// TwinCAT 3 PLC project x_template_xPlc
// Title: x_template_xPlc
// Company: TcOpen.MTS
// ProjectVersion: 0.6.0.913
// ProgramVersion: 3.1.4023.0
// libraries:
//   Tc2_Standard, * (Beckhoff Automation GmbH)
//   Tc2_System, * (Beckhoff Automation GmbH)
//   Tc3_Module, * (Beckhoff Automation GmbH)
//   TcoAbbRobotics, 0.11.0.68 (Vortex.Library)
//   TcoAbstractions, 0.11.0.68 (Vortex.Library)
//   TcoAimTtiPowerSupply, 0.11.0.68 (Vortex.Library)
//   TcoCognexVision, 0.11.0.68 (Vortex.Library)
//   TcoCore, 0.11.0.68 (Vortex.Library)
//   TcoData, 0.11.0.68 (Vortex.Library)
//   TcoDrivesBeckhoff, 0.11.0.68 (Vortex.Library)
//   TcoElements, 0.11.0.68 (Vortex.Library)
//   TcoInspectors, 0.11.0.68 (Vortex.Library)
//   TcoIo, 0.11.0.68 (Vortex.Library)
//   TcoKukaRobotics, 0.11.0.68 (Vortex.Library)
//   TcoMitsubishiRobotics, 0.11.0.68 (Vortex.Library)
//   TcoPneumatics, 0.11.0.68 (Vortex.Library)
//   TcoRexrothPress, 0.11.0.68 (Vortex.Library)
//   TcoTixonFeeding, 0.11.0.68 (Vortex.Library)
//   TcoUrRobotics, 0.11.0.68 (Vortex.Library)
//   TcoUtilities, 0.11.0.68 (Vortex.Library)
// project tree:
//   Abstractions/Components/ArrayRenderingExample/ SampleArrayToRender.TcDUT (not stored), SampleDataItem.TcDUT (not stored)
//   Abstractions/Components/MtsFeeding/ TcoFeedingSequenceTask.TcPOU, TcoPlsPaletizator.TcPOU, TcoPlsPaletizator_Components.TcDUT, TcoPlsPaletizator_Config_v_1_x_x.TcDUT, TcoPlsPaletizator_Control_v_1_x_x.TcDUT (not stored), TcoPlsPaletizator_Status_v_1_x_x.TcDUT
//   Abstractions/Components/WrappedComponent/ WrappedComponentExample.TcPOU (not stored), WrappedComponentExample_Config.TcDUT (not stored), WrappedComponentExample_Control.TcDUT (not stored), WrappedComponentExample_Status.TcDUT (not stored), WrappedComponentsExample.TcDUT (not stored)
//   Abstractions/CUBase/ CuBaseRecurringFail.TcDUT (not stored), CuBaseRecurringFailures.TcDUT (not stored), CUBase.TcPOU (not stored), CUBaseStatusInfo.TcDUT (not stored), CUBaseSettings.TcDUT (not stored), CUComponentsBase.TcDUT (not stored), ICUBase.TcIO (not stored), ICUTask.TcIO (not stored), OperatorInfo.TcDUT (not stored)
//   Abstractions/CUBase/Data/ CuHeader.TcDUT (not stored), CUProcessDataBase.TcDUT (not stored), CUTechnologicalDataBase.TcDUT (not stored), eCUMode.TcDUT (not stored), eCUState.TcDUT (not stored), eDataEntityInvokeType.TcDUT (not stored), EntityHeader.TcDUT (not stored)
//   Abstractions/CUBase/RemoteTasks/ ProductionPlaner.TcPOU (not stored)
//   Abstractions/CUBase/Tasks/ CUBaseAutomat.TcPOU (not stored), CUBaseSuspend.TcPOU (not stored), CUBaseGround.TcPOU (not stored), CUBaseRecover.TcPOU (not stored)
//   Abstractions/Generic/NotificationPanel/ NotificationPanel.TcPOU (not stored), NotificationPanelInfo.TcDUT (not stored)
//   Abstractions/Generic/TagsPairing/ eTagPairingAnswer.TcDUT (not stored), eTagPairingMode.TcDUT (not stored), eTagPairingStatus.TcDUT (not stored), PairTagTask.TcPOU (not stored), TagsPairing.TcDUT (not stored)
//   Abstractions/Safety/ControlButtons/ TcoControlButtons.TcPOU (not stored), ITcoControlButtons.TcIO (not stored), TcoControledZone_Info.TcDUT (not stored)
//   Abstractions/Safety/ControlledZone/ TcoControlledZoneActionTask.TcPOU (not stored), TcoControlledZone.TcPOU (not stored), TcoControlledZone_Config.TcDUT (not stored), TcoControlledZone_Status.TcDUT (not stored)
//   Abstractions/Safety/ControlVoltage/ ITcoControlVoltage.TcIO (not stored), TcoControlVoltage.TcPOU (not stored)
//   Abstractions/Safety/DoorCircuit/ TcoDoorCircuit_Status.TcDUT (not stored), TcoDoorCircuit_Config.TcDUT (not stored), TcoDoorCircuit.TcPOU (not stored), ITcoDoorCircuit.TcIO (not stored)
//   Abstractions/Safety/Doors/ ITcoDoorLock.TcIO (not stored), TcoStandardDoor.TcPOU (not stored), TcoBasicDoor.TcPOU (not stored)
//   Abstractions/Safety/Estop/ TcoEmergencyStop.TcPOU (not stored)
//   Abstractions/Safety/KeyMode/ TcoKeyMode_Config.TcDUT (not stored), TcoKeyMode_Status.TcDUT (not stored), TcoKeyMode.TcPOU (not stored), ITcoKeyMode.TcIO (not stored)
//   Abstractions/Safety/KeyNormalService/ TcoKeyNormalService.TcPOU (not stored), ITcoKeyNormalSevice.TcIO (not stored)
//   Abstractions/TcoCore/ CycleTimeAnalitics.TcDUT (not stored), TcoInnerTask.TcPOU (not stored), TcoTaskedSequencer.TcPOU (not stored), TcoTaskedService.TcPOU (not stored)
//   Abstractions/Technology/ eStations.TcDUT (not stored)
//   / MAIN.TcPOU (not stored), PlcTask.TcTTO (not stored)
//   Technology/CU00x/Automat/ CU00xAutomatParalell_1_Task.TcPOU (not stored), CU00xAutomatTask.TcPOU (not stored)
//   Technology/CU00x/Components/ CU00xExamplesOfComponents.TcDUT, CU00xComponents.TcDUT
//   Technology/CU00x/Data/ CU00xTechnologicalData.TcDUT (not stored), CU00xDialogContent.TcPOU (not stored), CU00xProcessData.TcDUT (not stored)
//   Technology/CU00x/Ground/ CU00xGroundTask.TcPOU (not stored)
//   Technology/CU00x/Manual/ CU00xManualTask.TcPOU (not stored)
//   Technology/CU00x/Positions/ CU00xTestMultiPositions.TcPOU (not stored), Cu00xTestPositions.TcPOU (not stored)
//   Technology/CU00x/Safety/Suspend/ CU00xSuspendTask.TcPOU
//   Technology/CU00x/Safety/Recover/ CU00xRecoverTask.TcPOU (not stored)
//   Technology/Data/ ProcessData.TcDUT, ProcessDataManager.TcPOU (not stored), TcoEntityBase.TcDUT, TechnologicalDataManager.TcPOU (not stored), TechnologyData.TcDUT
//   Technology/CU00x/ CU00x.TcPOU
//   Technology/ Technology.TcPOU, TechnologyComponents.TcDUT (not stored)
//   DUTs/IO/PDOs/ Device_State_F0482DC3.TcDUT, Device_Control_6258066A.TcDUT, Inputs_23559BB0.TcDUT, Outputs_FC2FACAD.TcDUT, Modules_85784B27.TcDUT, Channel_830843C1.TcDUT, Channel_42CA91F7.TcDUT
//   DUTs/IO/Boxes/ EK1200_013D0B49.TcDUT, EK1122_1FC0878B.TcDUT (not stored), AES_510494FB.TcDUT, EPP1322_1FC0878B.TcDUT, EPP1809_32157CFD.TcDUT, EPP1008_78E8D3DD.TcDUT, EL1809_32157CFD.TcDUT (not stored), EL2809_2B6483BD.TcDUT, EL9011_D65D3D32.TcDUT
//   DUTs/IO/Devices/ SyncUnitTasks_4BE01469.TcDUT, SyncUnits_67D36DDA.TcDUT
//   DUTs/IO/Topology/ EK_E812B8FA.TcDUT, EC_4E5C738F.TcDUT, EC_245FBB9A.TcDUT
//   GVLs/ GVL_iXlinker.TcGVL
// real-time tasks:
//   TASK PlcTask: cycle T#10ms, priority 20, ADS port 350
//   TASK PlcTask1: cycle T#10ms, priority 21, ADS port 351
// I/O:
//   DEVICE EC1 (disabled), AmsNetId 172.20.21.220.7.1
//     (EK1200) [EK1200-5000 EtherCAT Power supply (2A E-Bus)]
//       EC (EK1122) [EK1122 2 port EtherCAT junction]
//       PN (EL6631) [EL6631 PROFINET IO Controller]
//       IA1 (EL1809) [EL1809 16Ch. Dig. Input 24V, 3ms]
//       QA1 (EL2809) [EL2809 16Ch. Dig. Output 24V, 0.5A]
//       Term 6 (EL4004) [EL4004 4Ch. Ana. Output 0-10V, 12bit]
//       Term 7 (EL7342) [EL7342 2Ch. DC motor output stage (50V, 3.5A)]
//       Term 8 (EL4004) [EL4004 4Ch. Ana. Output 0-10V, 12bit]
//       Term 9 (EL6001) [EL6001 Interface (RS232)]
//       Term 13 (EL9011) [EL9011 End Terminal]
//   DEVICE EC (disabled), AmsNetId 172.20.21.220.2.1
//     EC [EK1200-5000 EtherCAT Power supply (2A E-Bus)]
//       EK [EK1122 2 port EtherCAT junction]
//         PNEU [AES Fieldbus Coupler Gen2]
//           modules: Modules
//         AB [EPP1322-0001 3 port EtherCAT P gateway]
//         AB21 [EPP1809-0021 16 Ch. Dig. Input 24V, 3ms, M8]
//         AB22 [EPP1809-0021 16 Ch. Dig. Input 24V, 3ms, M8]
//         AB23 [EPP1008-0001 8 Ch. Dig. Input 24V, 3ms, M8]
//         AB24 [EPP1008-0001 8 Ch. Dig. Input 24V, 3ms, M8]
//       IA1 [EL1809 16Ch. Dig. Input 24V, 3ms]
//       QA1 [EL2809-0015 16Ch. Dig. Output 24V DC, 0.35A, not short-circuit proof]
//       Term 11 (EL9011) [EL9011 End Terminal]
// variable links:
//   x_template_xPlc/x_template_xPlc Instance <-> EC
//     PlcTask Inputs/GVL_iXlinker.EC.InfoData.AmsNetId <-> InfoData/AmsNetId
//     PlcTask Inputs/GVL_iXlinker.EC.InfoData.CfgSlaveCount <-> InfoData/CfgSlaveCount
//     PlcTask Inputs/GVL_iXlinker.EC.InfoData.ChangeCount <-> InfoData/ChangeCount
//     PlcTask Inputs/GVL_iXlinker.EC.InfoData.DevId <-> InfoData/DevId
//     PlcTask Inputs/GVL_iXlinker.EC.Inputs.DevState <-> Inputs/DevState
//     PlcTask Inputs/GVL_iXlinker.EC.Inputs.Frm0InputToggle <-> Inputs/Frm0InputToggle
//     PlcTask Inputs/GVL_iXlinker.EC.Inputs.Frm0State <-> Inputs/Frm0State
//     PlcTask Inputs/GVL_iXlinker.EC.Inputs.Frm0WcState <-> Inputs/Frm0WcState
//     PlcTask Inputs/GVL_iXlinker.EC.Inputs.SlaveCount <-> Inputs/SlaveCount
//     PlcTask Inputs/GVL_iXlinker.EC.SyncUnits._default.PlcTask.InfoData.ObjectId <-> SyncUnits/<default>/PlcTask/InfoData/ObjectId
//     PlcTask Inputs/GVL_iXlinker.EC.SyncUnits._default.PlcTask.InfoData.SlaveCount <-> SyncUnits/<default>/PlcTask/InfoData/SlaveCount
//     PlcTask Inputs/GVL_iXlinker.EC.SyncUnits._default.PlcTask.InfoData.State <-> SyncUnits/<default>/PlcTask/InfoData/State
//     PlcTask Inputs/GVL_iXlinker.EC.SyncUnits._default.PlcTask.WcState.WcState <-> SyncUnits/<default>/PlcTask/WcState/WcState
//     PlcTask Outputs/GVL_iXlinker.EC.Outputs.DevCtrl <-> Outputs/DevCtrl
//     PlcTask Outputs/GVL_iXlinker.EC.Outputs.Frm0Ctrl <-> Outputs/Frm0Ctrl
//     PlcTask Outputs/GVL_iXlinker.EC.Outputs.Frm0WcCtrl <-> Outputs/Frm0WcCtrl
//   x_template_xPlc/x_template_xPlc Instance <-> EC/EC/EK
//     PlcTask Inputs/GVL_iXlinker.EC.EC.EK.InfoData.State <-> InfoData/State
//   x_template_xPlc/x_template_xPlc Instance <-> EC/EC/EK/AB
//     PlcTask Inputs/GVL_iXlinker.EC.EC.EK.AB.InfoData.State <-> InfoData/State
//   x_template_xPlc/x_template_xPlc Instance <-> EC/EC/EK/AB21
//     PlcTask Inputs/GVL_iXlinker.EC.EC.EK.AB21.Channel_{1..16}.Input <-> Channel {1..16}/Input  (16 links)
//     PlcTask Inputs/GVL_iXlinker.EC.EC.EK.AB21.InfoData.State <-> InfoData/State
//     PlcTask Inputs/GVL_iXlinker.EC.EC.EK.AB21.WcState.InputToggle <-> WcState/InputToggle
//     PlcTask Inputs/GVL_iXlinker.EC.EC.EK.AB21.WcState.WcState <-> WcState/WcState
//   x_template_xPlc/x_template_xPlc Instance <-> EC/EC/EK/AB22
//     PlcTask Inputs/GVL_iXlinker.EC.EC.EK.AB22.Channel_{1..16}.Input <-> Channel {1..16}/Input  (16 links)
//     PlcTask Inputs/GVL_iXlinker.EC.EC.EK.AB22.InfoData.State <-> InfoData/State
//     PlcTask Inputs/GVL_iXlinker.EC.EC.EK.AB22.WcState.InputToggle <-> WcState/InputToggle
//     PlcTask Inputs/GVL_iXlinker.EC.EC.EK.AB22.WcState.WcState <-> WcState/WcState
//   x_template_xPlc/x_template_xPlc Instance <-> EC/EC/EK/AB23
//     PlcTask Inputs/GVL_iXlinker.EC.EC.EK.AB23.Channel_{1..8}.Input <-> Channel {1..8}/Input  (8 links)
//     PlcTask Inputs/GVL_iXlinker.EC.EC.EK.AB23.InfoData.State <-> InfoData/State
//     PlcTask Inputs/GVL_iXlinker.EC.EC.EK.AB23.WcState.InputToggle <-> WcState/InputToggle
//     PlcTask Inputs/GVL_iXlinker.EC.EC.EK.AB23.WcState.WcState <-> WcState/WcState
//   x_template_xPlc/x_template_xPlc Instance <-> EC/EC/EK/AB24
//     PlcTask Inputs/GVL_iXlinker.EC.EC.EK.AB24.Channel_{1..8}.Input <-> Channel {1..8}/Input  (8 links)
//     PlcTask Inputs/GVL_iXlinker.EC.EC.EK.AB24.InfoData.State <-> InfoData/State
//     PlcTask Inputs/GVL_iXlinker.EC.EC.EK.AB24.WcState.InputToggle <-> WcState/InputToggle
//     PlcTask Inputs/GVL_iXlinker.EC.EC.EK.AB24.WcState.WcState <-> WcState/WcState
//   x_template_xPlc/x_template_xPlc Instance <-> EC/EC/EK/PNEU
//     PlcTask Inputs/GVL_iXlinker.EC.EC.EK.PNEU.Device_State.CommonValve <-> Device_State/CommonValve
//     PlcTask Inputs/GVL_iXlinker.EC.EC.EK.PNEU.Device_State.Configuration_Error_IO_Module <-> Device_State/Configuration Error IO-Module
//     PlcTask Inputs/GVL_iXlinker.EC.EC.EK.PNEU.Device_State.Configuration_Error_Valve <-> Device_State/Configuration Error Valve
//     PlcTask Inputs/GVL_iXlinker.EC.EC.EK.PNEU.Device_State.Configuratipn_Error_SLS <-> Device_State/Configuratipn Error SLS
//     PlcTask Inputs/GVL_iXlinker.EC.EC.EK.PNEU.Device_State.Count_IO_Module_to_big <-> Device_State/Count IO-Module to big
//     PlcTask Inputs/GVL_iXlinker.EC.EC.EK.PNEU.Device_State.Heardbeat_x <-> Device_State/Heardbeat
//     PlcTask Inputs/GVL_iXlinker.EC.EC.EK.PNEU.Device_State.IO_1_8 <-> Device_State/IO:1-8
//     PlcTask Inputs/GVL_iXlinker.EC.EC.EK.PNEU.Device_State.IO_9_10 <-> Device_State/IO:9-10
//     PlcTask Inputs/GVL_iXlinker.EC.EC.EK.PNEU.Device_State.Switchcounter_Error <-> Device_State/Switchcounter Error
//     PlcTask Inputs/GVL_iXlinker.EC.EC.EK.PNEU.Device_State.UA_OFF <-> Device_State/UA OFF
//     PlcTask Inputs/GVL_iXlinker.EC.EC.EK.PNEU.Device_State.UL_OFF <-> Device_State/UL OFF
//     PlcTask Inputs/GVL_iXlinker.EC.EC.EK.PNEU.Device_State.Undervoltage_5V <-> Device_State/Undervoltage 5V
//     PlcTask Inputs/GVL_iXlinker.EC.EC.EK.PNEU.Device_State.Undervoltage_UA <-> Device_State/Undervoltage UA
//     PlcTask Inputs/GVL_iXlinker.EC.EC.EK.PNEU.Device_State.Undervoltage_UL <-> Device_State/Undervoltage UL
//     PlcTask Inputs/GVL_iXlinker.EC.EC.EK.PNEU.Device_State.Unknown_Module_ID <-> Device_State/Unknown Module ID
//     PlcTask Inputs/GVL_iXlinker.EC.EC.EK.PNEU.Device_State.ValveExtSupplyDiag_1_6 <-> Device_State/ValveExtSupplyDiag:1-6
//     PlcTask Inputs/GVL_iXlinker.EC.EC.EK.PNEU.InfoData.AdsAddr <-> InfoData/AdsAddr
//     PlcTask Inputs/GVL_iXlinker.EC.EC.EK.PNEU.InfoData.State <-> InfoData/State
//     PlcTask Inputs/GVL_iXlinker.EC.EC.EK.PNEU.Modules.Inputs.digital_Data_I[{0..31}] <-> Modules/Inputs/digital Data I_{0..31}  (32 links)
//     PlcTask Inputs/GVL_iXlinker.EC.EC.EK.PNEU.WcState.InputToggle <-> WcState/InputToggle
//     PlcTask Inputs/GVL_iXlinker.EC.EC.EK.PNEU.WcState.WcState <-> WcState/WcState
//     PlcTask Outputs/GVL_iXlinker.EC.EC.EK.PNEU.Device_Control.Default_Modul_Control <-> Device_Control/Default_Modul_Control
//     PlcTask Outputs/GVL_iXlinker.EC.EC.EK.PNEU.Device_Control.Freeze_Output <-> Device_Control/Freeze Output
//     PlcTask Outputs/GVL_iXlinker.EC.EC.EK.PNEU.Device_Control.HL_Swap <-> Device_Control/HL_Swap
//     PlcTask Outputs/GVL_iXlinker.EC.EC.EK.PNEU.Device_Control.Web_App_Disable <-> Device_Control/Web App Disable
//     PlcTask Outputs/GVL_iXlinker.EC.EC.EK.PNEU.Modules.Outputs.digital_Data_O[{0..31}] <-> Modules/Outputs/digital Data O_{0..31}  (32 links)
//   x_template_xPlc/x_template_xPlc Instance <-> EC/EC/IA1
//     PlcTask Inputs/GVL_iXlinker.EC.EC.IA1.Channel_{1..16}.Input <-> Channel {1..16}/Input  (16 links)
//     PlcTask Inputs/GVL_iXlinker.EC.EC.IA1.InfoData.State <-> InfoData/State
//     PlcTask Inputs/GVL_iXlinker.EC.EC.IA1.WcState.InputToggle <-> WcState/InputToggle
//     PlcTask Inputs/GVL_iXlinker.EC.EC.IA1.WcState.WcState <-> WcState/WcState
//   x_template_xPlc/x_template_xPlc Instance <-> EC/EC/QA1
//     PlcTask Inputs/GVL_iXlinker.EC.EC.QA1.InfoData.State <-> InfoData/State
//     PlcTask Inputs/GVL_iXlinker.EC.EC.QA1.WcState.WcState <-> WcState/WcState
//     PlcTask Outputs/GVL_iXlinker.EC.EC.QA1.Channel_{1..16}.Output <-> Channel {1..16}/Output  (16 links)

// ---- Abstractions/Components/MtsFeeding/TcoPlsPaletizator_Components.TcDUT
TYPE TcoPlsPaletizator_Components EXTENDS TcoCore.TcoStruct:
STRUCT
	
	{attribute wpf [Container(Layout.Stack)]}
	{attribute addProperty Name "(I1) <#Pritomnost blistra v presuvaci#>"}
	I1_PresentBlisterEntry : TcoElements.TcoDi(THISSTRUCT);
	
	{attribute addProperty Name "(I2) <#Pritomnost medzery medzi blistrami#>"}
	I2_PresentBlisterEntryEmptySpace : TcoElements.TcoDi(THISSTRUCT);
	
	{attribute addProperty Name "(I3) <#Zasobik blistrov prazdny#>"}
	I3_PresentBlistersInBufferEmpty : TcoElements.TcoDi(THISSTRUCT);

	
	{attribute addProperty Name "(I4) <#Pritomnost blistra v pracovnej pozicii#>"}
	I4_PresentBlisterInWorkingPos : TcoElements.TcoDi(THISSTRUCT);
	
	
	{attribute addProperty Name "(I5) <#Vystupny blister neje v sklzovom dopravniku#>"}
	I5_OutBlistersIsThrowedCorrectly : TcoElements.TcoDi(THISSTRUCT);
	
	{attribute addProperty Name "(I6) <#Vystupny blister snimanie vo vytahu#>"}
	I6_OutBlistersLisftSignal : TcoElements.TcoDi(THISSTRUCT);
	
	{attribute addProperty Name "(I7) <#Vystupny blister je nad Bufferom#>"}
	I7_OutBlistersIsAboveOutBuffer : TcoElements.TcoDi(THISSTRUCT);
	
	{attribute addProperty Name "(I8) <#Vystupny zasobnik je plny#>"}
	I8_OutBlistersBufferIsFull : TcoElements.TcoDi(THISSTRUCT);
	
	
	{attribute wpf [Container(Layout.Stack)]}
	{attribute addProperty Name "(P1) <#Vertikalny prisun vstupnych blistrov#>"}
	P1_VerticalSepareEntryBlisters : TcoPneumatics.TcoCylinder(THISSTRUCT);
	
	{attribute addProperty Name "(P2) <#Vertikalny prisun vstupnych blistrov #>"}
	P2_VerticalSepareEntryBlisters : TcoPneumatics.TcoCylinder(THISSTRUCT);
	
	{attribute addProperty Name "(P3) (P3.1) <#Horizontalny prisun vstupnych blistrov#>"}
	P3_HorizontalSepareEntryBlisters : TcoPneumatics.TcoDoubleCylinder(THISSTRUCT);
		
	{attribute addProperty Name "(P4) <#Prisun vstupneho blistra#>"}
	P4_FeedEntryBlister :TcoPneumatics.TcoCylinder(THISSTRUCT);
	
	{attribute addProperty Name "(P5) (P5.1)<#Horizontalny prisun vystupnych blistrov#>"}
	P5_HorizontalSepareOutBlisters : TcoPneumatics.TcoDoubleCylinder(THISSTRUCT);
	
	{attribute addProperty Name "(P6)<#Vertikalny prisun vystupnych blistrov#>"}
	P6_VerticalSepareOutBlister : TcoPneumatics.TcoCylinder(THISSTRUCT);
	
	{attribute addProperty Name "(P7) <#Podopretie vstupneho blistra#>"}
	P7_SupportEntryBlister : TcoPneumatics.TcoCylinder(THISSTRUCT);
	
	{attribute addProperty Name "(P8) (P8.1) <#Upevnenie zboku vstupneho blistra#>"}
	P8_FixEntryBlisterSide : TcoPneumatics.TcoDoubleCylinder(THISSTRUCT);
	
	{attribute addProperty Name "(P9) (P9.1) <#Zamknutue zhora vstupneho blistra#>"}
	P9_LockEntryBlisterTop : TcoPneumatics.TcoDoubleCylinder(THISSTRUCT);
	
	{attribute addProperty Name "(P10) (P10.1)<#Odelovac blistrov na vstupe#>"}
	P10_HoldEntrySepareOutBlister : TcoPneumatics.TcoDoubleCylinder(THISSTRUCT);
	
	
	
	{attribute wpf [Container(Layout.Stack,"Vseobecne")]}
	
	{attribute addProperty Name "(Q1) <#Signalizacia upozornenia R#>"}
	Q1_AttentionSignalisationR : TcoElements.TcoDo(THISSTRUCT);
	{attribute addProperty Name "(Q2) <#Signalizacia upozornenia G#>"}
	Q2_AttentionSignalisationG : TcoElements.TcoDo(THISSTRUCT);
	{attribute addProperty Name "(Q3) <#Signalizacia upozornenia B#>"}
	Q3_AttentionSignalisationB : TcoElements.TcoDo(THISSTRUCT);

	
	
END_STRUCT
END_TYPE

// ---- Abstractions/Components/MtsFeeding/TcoPlsPaletizator_Config_v_1_x_x.TcDUT
TYPE
    TcoPlsPaletizator_Config_v_1_x_x EXTENDS TcoCore.TcoStruct :
    STRUCT

	
        {attribute addProperty Name "<#Stabilizacny cas#>"}
		StabilisationTime : TIME :=T#500MS;
		{attribute addProperty Name "<#Blink period#> "}
		BlinkTime : TIME := T#500MS;
		
        {attribute addProperty Name "<#Zamykanie blistra zhora neaktive (P9)(P9.1)je nepritomne#>"}
		LockBlisterInPickPosInactive : BOOL;
		
		{attribute addProperty Name "<#Oddelovanie blistrov na vstupe neaktive (P10)(P10.1)je nepritomne#>"}
		SepareBlistersAtEntryInactive : BOOL;
    END_STRUCT
END_TYPE

// ---- Abstractions/Components/MtsFeeding/TcoPlsPaletizator_Status_v_1_x_x.TcDUT
TYPE
    TcoPlsPaletizator_Status_v_1_x_x EXTENDS TcoCore.TcoStruct :
    STRUCT

        ActionDescription : STRING;
        SafeCondition : BOOL;
		EntryBufferEmpty:BOOL;
        BlisterReady : BOOL;
        OutBufferFull : BOOL;
    END_STRUCT
END_TYPE

// ---- Technology/CU00x/Components/CU00xExamplesOfComponents.TcDUT
{attribute wpf [Container(Layout.Stack)]}	
{attribute wpf [Group(Layout.Scroll)]}
TYPE CU00xExamplesOfComponents EXTENDS TcoCore.TcoStruct:
STRUCT
		{attribute wpf [Container(Layout.Stack,"PNEU")]}	
		{attribute addProperty Name "(A1)HORIZONTAL AXIS"}
      	horizontalCylinder : TcoPneumatics.TcoCylinder(THISSTRUCT); 
		{attribute addProperty Name "(A2)VERTICAL AXIS"}
      	verticalCylinder : TcoPneumatics.TcoCylinder(THISSTRUCT); 
		
		{attribute addProperty Name "(A3)DOUBLE "}
      	doubleCylinder : TcoPneumatics.TcoDoubleCylinder(THISSTRUCT); 
		
		{attribute wpf [Container(Layout.Stack,"INPUTS")]}	
		{attribute addProperty Name "PRESENCE ON INSPECTION"}
     	PresenceOnInspection : TcoElements.TcoDi(THISSTRUCT);
		
		{attribute addProperty Name "PRESENCE AT ENTRY CONVEYOR"}
     	PresenceComponentAtEntr: TcoElements.TcoDi(THISSTRUCT);
		
		{attribute addProperty Name "COLISION SENSOR"}
     	ColisonSensorComponent: TcoElements.TcoDi(THISSTRUCT);

		{attribute addProperty Name "CONVEYOR AT ENTRY IS EMPTY"}
     	ConvAtEntryIsEmpty : TcoElements.TcoDi(THISSTRUCT);
		
		{attribute addProperty Name "INSPECTION NOK"}
     	InspectionIsNok : TcoElements.TcoDi(THISSTRUCT);
		

		{attribute wpf [Container(Layout.Stack,"OUTPUTS")]}		
		{attribute addProperty Name "LIGHT ON"}
     	LightOn : TcoElements.TcoDi(THISSTRUCT); 
		
		{attribute addProperty Name "LIGHT OFF"}
     	LightOff : TcoElements.TcoDi(THISSTRUCT);
		{attribute wpf [Container(Layout.Stack,"ANALOGS")]}	
		{attribute addProperty Name "VERIFY SETPOINT"}
     	VerifySetpoint : TcoElements.TcoAi(THISSTRUCT);
		{attribute addProperty Name "SETPOINT"}
     	Setpoint : TcoElements.TcoAo(THISSTRUCT);   
		
		{attribute addProperty Name "SampleDataToRender"}
     	ArrayToRender : SampleArrayToRender;   
		
		

END_STRUCT
END_TYPE

// ---- Technology/Data/ProcessData.TcDUT
{attribute clr [Container(Layout.Tabs)]}
TYPE
    ProcessData EXTENDS TcoEntityBase :
    STRUCT
        {attribute addProperty Name "<#Entity header#>"}
        EntityHeader : EntityHeader     := (Parent := THISSTRUCT);
		{attribute addProperty Name "<#CU00x#>"}
		{attribute clr [Container(Layout.Stack)]}
        CU00x : CU00xProcessData := (Parent := THISSTRUCT);

    END_STRUCT
END_TYPE

// ---- Technology/CU00x/Components/CU00xComponents.TcDUT
{attribute wpf [Container(Layout.Tabs)]}

TYPE
    CU00xComponents EXTENDS CUComponentsBase :
    STRUCT

		{attribute wpf [Container(Layout.Stack)]}
		{attribute wpf [Group(Layout.Scroll)]}
		{attribute addProperty Name "Supplu TTI QL"}
     	Supply : TcoAimTtiPowerSupply.TcoQl355P_v_1_x_x (THISSTRUCT);
		{attribute wpf [Container(Layout.Stack)]}
		PairTagTask: PairTagTask(THISSTRUCT);
		{attribute wpf [Container(Layout.Stack,"DRIVES AND MANIPULATORS")]}	
		{attribute wpf [Group(Layout.Scroll)]}
		{attribute addProperty Name "MultiAxis"}
     	MultiAxis : TcoDrivesBeckhoff.TcoMultiAxis (THISSTRUCT);
		{attribute addProperty Name "Single Axis"}
     	SingleAxis : TcoDrivesBeckhoff.TcoSingleAxis (THISSTRUCT);
		{attribute addProperty Name "Simple drive"}
     	SimpleDrive : TcoDrivesBeckhoff.TcoDriveSimple (THISSTRUCT);


	
		{attribute wpf [Container(Layout.Stack,"ROBOTICS")]}	
		{attribute wpf [Group(Layout.Scroll)]}
		{attribute addProperty Name "Abb IRC 5"}
     	AbbIrc5 : TcoAbbRobotics.TcoIrc5_v_1_x_x (THISSTRUCT);
		{attribute addProperty Name "Abb Omnicore"}
     	AbbOmnicore : TcoAbbRobotics.TcoOmnicore_v_1_x_x (THISSTRUCT);
		
		{attribute addProperty Name "Mitshubishi Cr series"}
     	MitshubishiCr: TcoMitsubishiRobotics.TcoCr800_v_1_x_x (THISSTRUCT);
		{attribute addProperty Name "UR CB series"}
     	UrCb3:  TcoUrRobotics.TcoUrCb3_v_3_x_x(THISSTRUCT);
		{attribute addProperty Name "Ur E series"}
     	UrEseries: TcoUrRobotics.TcoUrEseries_v_5_x_x (THISSTRUCT);
		
		{attribute addProperty Name "Kuka Krc4"}
     	KukaKrc4: TcoKukaRobotics.TcoKrc4_v_5_x_x (THISSTRUCT);
		
		{attribute wpf [Container(Layout.Stack,"TIXONS")]}	
		{attribute wpf [Group(Layout.Scroll)]}
		{attribute addProperty Name "Tixon Vibro"}
     	TixonVibro : TcoTixonFeeding.TcoTixonVibro_v_1_x_x (THISSTRUCT);
		{attribute addProperty Name "Tixon Step"}
     	TixonStep : TcoTixonFeeding.TcoTixonStep_v_1_x_x(THISSTRUCT);
		
		{attribute addProperty Name "Tixon Pick Vibro"}
     	TixonPickVibro : TcoTixonFeeding.TcoTixonPickVibro_v_1_x_x (THISSTRUCT);
		{attribute addProperty Name "Tixon Pick Step"}
     	TixonPickStep : TcoTixonFeeding.TcoTixonPickStep_v_1_x_x(THISSTRUCT);
			
		{attribute wpf [Container(Layout.Stack,"MtsFeeding")]}	
		{attribute wpf [Group(Layout.Scroll)]}
		PlsPaletizator:TcoPlsPaletizator(THISSTRUCT);	
		{attribute clr [RenderIgnore()]}
		PlsPaletizatorComponents:TcoPlsPaletizator_Components:= (Parent := THISSTRUCT);  
		
		{attribute wpf [Container(Layout.Stack,"Wrapped component example")]}	
		{attribute wpf [Group(Layout.Scroll)]}
		PickAndPlace:WrappedComponentExample(THISSTRUCT);
		{attribute wpf [Container(Layout.Stack,"Wrapped component struct")]}	
		PickAndPlaceCompoennts:WrappedComponentsExample:= (Parent := THISSTRUCT);  

		{attribute addProperty Name "GROUP 1"}
		Group1 : CU00xExamplesOfComponents:= (Parent := THISSTRUCT);  
		{attribute addProperty Name "GROUP 2"}
		Group2 : CU00xExamplesOfComponents:= (Parent := THISSTRUCT); 
 
		
		
		
    END_STRUCT
END_TYPE

// ---- Technology/Data/TcoEntityBase.TcDUT
TYPE TcoEntityBase EXTENDS TcoData.TcoEntity :
STRUCT
	{attribute clr [RenderIgnore("Control", "ShadowControl")]}
	{attribute addProperty Name "<#Created#>"}
	_Created : DT;
	{attribute clr [RenderIgnore("Control", "ShadowControl")]}
	{attribute addProperty Name "<#Modified#>"}
	_Modified : DT;
	
END_STRUCT
END_TYPE

// ---- Technology/Data/TechnologyData.TcDUT
{attribute clr [Container(Layout.Tabs)]}
TYPE
    TechnologyData EXTENDS TcoEntityBase :
    STRUCT
        CU00x : CU00xTechnologicalData := (Parent := THISSTRUCT);
    END_STRUCT
END_TYPE

// ---- DUTs/IO/PDOs/Device_State_F0482DC3.TcDUT
{attribute 'GeneratedUsingTerminal: AES-D-BC-ECAT Gen2-0001'}
{attribute addProperty BoxType "AES-D-BC-ECAT Gen2-0001"}
{attribute addProperty Id "IO_1_8AT %I*BYTE1IO_9_10AT %I*BYTE1ValveExtSupplyDiag_1_6AT %I*BYTE1Undervoltage_UAAT %I*BOOL1UA_OFFAT %I*BOOL1Undervoltage_ULAT %I*BOOL1UL_OFFAT %I*BOOL1Undervoltage_5VAT %I*BOOL1CommonValveAT %I*BOOL1Configuration_Error_ValveAT %I*BOOL1Configuration_Error_IO_ModuleAT %I*BOOL1Switchcounter_ErrorAT %I*BOOL1Configuratipn_Error_SLSAT %I*BOOL1Heardbeat_xAT %I*BOOL1Unknown_Module_IDAT %I*BOOL1Count_IO_Module_to_bigAT %I*BOOL1"}
{attribute addProperty CRC "4031262147"}
{attribute addProperty Size "16"}
TYPE Device_State_F0482DC3 EXTENDS TcoIo.InputBase_8311D824 :
STRUCT
	{attribute addProperty Name "IO_1_8"}
	IO_1_8 AT %I* : BYTE;
	{attribute addProperty Name "IO_9_10"}
	IO_9_10 AT %I* : BYTE;
	{attribute addProperty Name "ValveExtSupplyDiag_1_6"}
	ValveExtSupplyDiag_1_6 AT %I* : BYTE;
	{attribute addProperty Name "Undervoltage_UA"}
	Undervoltage_UA AT %I* : BOOL;
	{attribute addProperty Name "UA_OFF"}
	UA_OFF AT %I* : BOOL;
	{attribute addProperty Name "Undervoltage_UL"}
	Undervoltage_UL AT %I* : BOOL;
	{attribute addProperty Name "UL_OFF"}
	UL_OFF AT %I* : BOOL;
	{attribute addProperty Name "Undervoltage_5V"}
	Undervoltage_5V AT %I* : BOOL;
	{attribute addProperty Name "CommonValve"}
	CommonValve AT %I* : BOOL;
	{attribute addProperty Name "Configuration_Error_Valve"}
	Configuration_Error_Valve AT %I* : BOOL;
	{attribute addProperty Name "Configuration_Error_IO_Module"}
	Configuration_Error_IO_Module AT %I* : BOOL;
	{attribute addProperty Name "Switchcounter_Error"}
	Switchcounter_Error AT %I* : BOOL;
	{attribute addProperty Name "Configuratipn_Error_SLS"}
	Configuratipn_Error_SLS AT %I* : BOOL;
	{attribute addProperty Name "Heardbeat_x"}
	Heardbeat_x AT %I* : BOOL;
	{attribute addProperty Name "Unknown_Module_ID"}
	Unknown_Module_ID AT %I* : BOOL;
	{attribute addProperty Name "Count_IO_Module_to_big"}
	Count_IO_Module_to_big AT %I* : BOOL;
END_STRUCT
END_TYPE

// ---- DUTs/IO/PDOs/Device_Control_6258066A.TcDUT
{attribute 'GeneratedUsingTerminal: AES-D-BC-ECAT Gen2-0001'}
{attribute addProperty BoxType "AES-D-BC-ECAT Gen2-0001"}
{attribute addProperty Id "Web_App_DisableAT %Q*BOOL1Freeze_OutputAT %Q*BOOL1HL_SwapAT %Q*BOOL1Default_Modul_ControlAT %Q*BOOL1"}
{attribute addProperty CRC "1649935978"}
{attribute addProperty Size "4"}
TYPE Device_Control_6258066A EXTENDS TcoIo.OutputBase_10CEE7DE :
STRUCT
	{attribute addProperty Name "Web_App_Disable"}
	Web_App_Disable AT %Q* : BOOL;
	{attribute addProperty Name "Freeze_Output"}
	Freeze_Output AT %Q* : BOOL;
	{attribute addProperty Name "HL_Swap"}
	HL_Swap AT %Q* : BOOL;
	{attribute addProperty Name "Default_Modul_Control"}
	Default_Modul_Control AT %Q* : BOOL;
END_STRUCT
END_TYPE

// ---- DUTs/IO/PDOs/Inputs_23559BB0.TcDUT
{attribute 'GeneratedUsingTerminal: AES-D-BC-ECAT Gen2-0001'}
{attribute addProperty BoxType "AES-D-BC-ECAT Gen2-0001"}
{attribute addProperty Id "digital_Data_IAT %I*ARRAY[0..31] OF USINT32"}
{attribute addProperty CRC "1374483313"}
{attribute addProperty Size "32"}
TYPE Inputs_23559BB0 EXTENDS TcoIo.InputBase_8311D824 :
STRUCT
	{attribute addProperty Name "digital_Data_I"}
	digital_Data_I AT %I* : ARRAY[0..31] OF USINT;
END_STRUCT
END_TYPE

// ---- DUTs/IO/PDOs/Outputs_FC2FACAD.TcDUT
{attribute 'GeneratedUsingTerminal: AES-D-BC-ECAT Gen2-0001'}
{attribute addProperty BoxType "AES-D-BC-ECAT Gen2-0001"}
{attribute addProperty Id "digital_Data_OAT %Q*ARRAY[0..31] OF USINT32"}
{attribute addProperty CRC "2024821696"}
{attribute addProperty Size "32"}
TYPE Outputs_FC2FACAD EXTENDS TcoIo.OutputBase_10CEE7DE :
STRUCT
	{attribute addProperty Name "digital_Data_O"}
	digital_Data_O AT %Q* : ARRAY[0..31] OF USINT;
END_STRUCT
END_TYPE

// ---- DUTs/IO/PDOs/Modules_85784B27.TcDUT
{attribute 'GeneratedUsingTerminal: AES-D-BC-ECAT Gen2-0001'}
{attribute addProperty BoxType "AES-D-BC-ECAT Gen2-0001"}
{attribute addProperty Id "InputsInputs_23559BB032OutputsOutputs_FC2FACAD32"}
{attribute addProperty CRC "2239253287"}
{attribute addProperty Size "64"}
TYPE Modules_85784B27 :
STRUCT
	{attribute addProperty Name "Inputs"}
	Inputs  : Inputs_23559BB0;
	{attribute addProperty Name "Outputs"}
	Outputs  : Outputs_FC2FACAD;
END_STRUCT
END_TYPE

// ---- DUTs/IO/PDOs/Channel_830843C1.TcDUT
{attribute 'GeneratedUsingTerminal: EPP1809-0021-0016'}
{attribute addProperty BoxType "EPP1809-0021-0016"}
{attribute addProperty Id "InputAT %I*BOOL1"}
{attribute addProperty CRC "2198356929"}
{attribute addProperty Size "1"}
TYPE Channel_830843C1 EXTENDS TcoIo.InputBase_8311D824 :
STRUCT
	{attribute addProperty Name "Input"}
	Input AT %I* : BOOL;
END_STRUCT
END_TYPE

// ---- DUTs/IO/PDOs/Channel_42CA91F7.TcDUT
{attribute 'GeneratedUsingTerminal: EL2809-0015-0016'}
{attribute addProperty BoxType "EL2809-0015-0016"}
{attribute addProperty Id "OutputAT %Q*BOOL1"}
{attribute addProperty CRC "1120571895"}
{attribute addProperty Size "1"}
TYPE Channel_42CA91F7 EXTENDS TcoIo.OutputBase_10CEE7DE :
STRUCT
	{attribute addProperty Name "Output"}
	Output AT %Q* : BOOL;
END_STRUCT
END_TYPE

// ---- DUTs/IO/Boxes/EK1200_013D0B49.TcDUT
{attribute 'GeneratedUsingTerminal: EK1200-1388-0000'}
{attribute addProperty VendorId "#x00000002"}
{attribute addProperty BoxType "EK1200-1388-0000"}
{attribute addProperty Description "EK1200-5000 EtherCAT Power supply (2A E-Bus)"}
{attribute addProperty Physics "YK"}
{attribute addProperty Id "EK1200"}
{attribute addProperty CRC "20777801"}
{attribute addProperty Size "0"}
TYPE EK1200_013D0B49 EXTENDS TcoIo.EtcSlaveBoxBase_77A0E4A7 :
STRUCT
END_STRUCT
END_TYPE

// ---- DUTs/IO/Boxes/AES_510494FB.TcDUT
{attribute 'GeneratedUsingTerminal: AES-D-BC-ECAT Gen2-0001'}
{attribute addProperty VendorId "#x000001b2"}
{attribute addProperty BoxType "AES-D-BC-ECAT Gen2-0001"}
{attribute addProperty Description "AES Fieldbus Coupler Gen2"}
{attribute addProperty Physics "YY"}
{attribute addProperty Id "ModulesModules_85784B2764Device_StateAT %I*Device_State_F0482DC316Device_ControlAT %Q*Device_Control_6258066A4WcStateAT %I*WcState_9091E0EB2InfoDataAT %I*InfoData_23CBA8372"}
{attribute addProperty CRC "1359254779"}
{attribute addProperty Size "88"}
TYPE AES_510494FB EXTENDS TcoIo.EtcSlaveBoxBase_77A0E4A7 :
STRUCT
	{attribute addProperty Name "Modules"}
	Modules : Modules_85784B27;
	{attribute addProperty Name "Device_State"}
	Device_State : Device_State_F0482DC3;
	{attribute addProperty Name "Device_Control"}
	Device_Control : Device_Control_6258066A;
	{attribute addProperty Name "WcState"}
	WcState : TcoIo.WcState_9091E0EB;
	{attribute addProperty Name "InfoData"}
	InfoData : TcoIo.InfoData_23CBA837;
END_STRUCT
END_TYPE

// ---- DUTs/IO/Boxes/EPP1322_1FC0878B.TcDUT
{attribute 'GeneratedUsingTerminal: EPP1322-0001-0017'}
{attribute addProperty VendorId "#x00000002"}
{attribute addProperty BoxType "EPP1322-0001-0017"}
{attribute addProperty Description "EPP1322-0001 3 port EtherCAT P gateway"}
{attribute addProperty Physics "YYYY"}
{attribute addProperty Id "InfoDataAT %I*InfoData_6F19DB2B2"}
{attribute addProperty CRC "532711307"}
{attribute addProperty Size "2"}
TYPE EPP1322_1FC0878B EXTENDS TcoIo.EtcSlaveBoxBase_77A0E4A7 :
STRUCT
	{attribute addProperty Name "InfoData"}
	InfoData : TcoIo.InfoData_6F19DB2B;
END_STRUCT
END_TYPE

// ---- DUTs/IO/Boxes/EPP1809_32157CFD.TcDUT
{attribute 'GeneratedUsingTerminal: EPP1809-0021-0016'}
{attribute addProperty VendorId "#x00000002"}
{attribute addProperty BoxType "EPP1809-0021-0016"}
{attribute addProperty Description "EPP1809-0021 16 Ch. Dig. Input 24V, 3ms, M8"}
{attribute addProperty Physics "YY"}
{attribute addProperty Id "Channel_1AT %I*Channel_830843C11Channel_2AT %I*Channel_830843C11Channel_3AT %I*Channel_830843C11Channel_4AT %I*Channel_830843C11Channel_5AT %I*Channel_830843C11Channel_6AT %I*Channel_830843C11Channel_7AT %I*Channel_830843C11Channel_8AT %I*Channel_830843C11Channel_9AT %I*Channel_830843C11Channel_10AT %I*Channel_830843C11Channel_11AT %I*Channel_830843C11Channel_12AT %I*Channel_830843C11Channel_13AT %I*Channel_830843C11Channel_14AT %I*Channel_830843C11Channel_15AT %I*Channel_830843C11Channel_16AT %I*Channel_830843C11WcStateAT %I*WcState_9091E0EB2InfoDataAT %I*InfoData_6F19DB2B2"}
{attribute addProperty CRC "840269053"}
{attribute addProperty Size "20"}
TYPE EPP1809_32157CFD EXTENDS TcoIo.EtcSlaveBoxBase_77A0E4A7 :
STRUCT
	{attribute addProperty Name "Channel_1"}
	Channel_1 : Channel_830843C1;
	{attribute addProperty Name "Channel_2"}
	Channel_2 : Channel_830843C1;
	{attribute addProperty Name "Channel_3"}
	Channel_3 : Channel_830843C1;
	{attribute addProperty Name "Channel_4"}
	Channel_4 : Channel_830843C1;
	{attribute addProperty Name "Channel_5"}
	Channel_5 : Channel_830843C1;
	{attribute addProperty Name "Channel_6"}
	Channel_6 : Channel_830843C1;
	{attribute addProperty Name "Channel_7"}
	Channel_7 : Channel_830843C1;
	{attribute addProperty Name "Channel_8"}
	Channel_8 : Channel_830843C1;
	{attribute addProperty Name "Channel_9"}
	Channel_9 : Channel_830843C1;
	{attribute addProperty Name "Channel_10"}
	Channel_10 : Channel_830843C1;
	{attribute addProperty Name "Channel_11"}
	Channel_11 : Channel_830843C1;
	{attribute addProperty Name "Channel_12"}
	Channel_12 : Channel_830843C1;
	{attribute addProperty Name "Channel_13"}
	Channel_13 : Channel_830843C1;
	{attribute addProperty Name "Channel_14"}
	Channel_14 : Channel_830843C1;
	{attribute addProperty Name "Channel_15"}
	Channel_15 : Channel_830843C1;
	{attribute addProperty Name "Channel_16"}
	Channel_16 : Channel_830843C1;
	{attribute addProperty Name "WcState"}
	WcState : TcoIo.WcState_9091E0EB;
	{attribute addProperty Name "InfoData"}
	InfoData : TcoIo.InfoData_6F19DB2B;
END_STRUCT
END_TYPE

// ---- DUTs/IO/Boxes/EPP1008_78E8D3DD.TcDUT
{attribute 'GeneratedUsingTerminal: EPP1008-0001-0017'}
{attribute addProperty VendorId "#x00000002"}
{attribute addProperty BoxType "EPP1008-0001-0017"}
{attribute addProperty Description "EPP1008-0001 8 Ch. Dig. Input 24V, 3ms, M8"}
{attribute addProperty Physics "YY"}
{attribute addProperty Id "Channel_1AT %I*Channel_830843C11Channel_2AT %I*Channel_830843C11Channel_3AT %I*Channel_830843C11Channel_4AT %I*Channel_830843C11Channel_5AT %I*Channel_830843C11Channel_6AT %I*Channel_830843C11Channel_7AT %I*Channel_830843C11Channel_8AT %I*Channel_830843C11WcStateAT %I*WcState_9091E0EB2InfoDataAT %I*InfoData_6F19DB2B2"}
{attribute addProperty CRC "2028524509"}
{attribute addProperty Size "12"}
TYPE EPP1008_78E8D3DD EXTENDS TcoIo.EtcSlaveBoxBase_77A0E4A7 :
STRUCT
	{attribute addProperty Name "Channel_1"}
	Channel_1 : Channel_830843C1;
	{attribute addProperty Name "Channel_2"}
	Channel_2 : Channel_830843C1;
	{attribute addProperty Name "Channel_3"}
	Channel_3 : Channel_830843C1;
	{attribute addProperty Name "Channel_4"}
	Channel_4 : Channel_830843C1;
	{attribute addProperty Name "Channel_5"}
	Channel_5 : Channel_830843C1;
	{attribute addProperty Name "Channel_6"}
	Channel_6 : Channel_830843C1;
	{attribute addProperty Name "Channel_7"}
	Channel_7 : Channel_830843C1;
	{attribute addProperty Name "Channel_8"}
	Channel_8 : Channel_830843C1;
	{attribute addProperty Name "WcState"}
	WcState : TcoIo.WcState_9091E0EB;
	{attribute addProperty Name "InfoData"}
	InfoData : TcoIo.InfoData_6F19DB2B;
END_STRUCT
END_TYPE

// ---- DUTs/IO/Boxes/EL2809_2B6483BD.TcDUT
{attribute 'GeneratedUsingTerminal: EL2809-0015-0016'}
{attribute addProperty VendorId "#x00000002"}
{attribute addProperty BoxType "EL2809-0015-0016"}
{attribute addProperty Description "EL2809-0015 16Ch. Dig. Output 24V DC, 0.35A, not short-circuit proof"}
{attribute addProperty Physics "KK"}
{attribute addProperty Id "Channel_1AT %Q*Channel_42CA91F71Channel_2AT %Q*Channel_42CA91F71Channel_3AT %Q*Channel_42CA91F71Channel_4AT %Q*Channel_42CA91F71Channel_5AT %Q*Channel_42CA91F71Channel_6AT %Q*Channel_42CA91F71Channel_7AT %Q*Channel_42CA91F71Channel_8AT %Q*Channel_42CA91F71Channel_9AT %Q*Channel_42CA91F71Channel_10AT %Q*Channel_42CA91F71Channel_11AT %Q*Channel_42CA91F71Channel_12AT %Q*Channel_42CA91F71Channel_13AT %Q*Channel_42CA91F71Channel_14AT %Q*Channel_42CA91F71Channel_15AT %Q*Channel_42CA91F71Channel_16AT %Q*Channel_42CA91F71WcStateAT %I*WcState_0B2B16F91InfoDataAT %I*InfoData_6F19DB2B2"}
{attribute addProperty CRC "728007613"}
{attribute addProperty Size "19"}
TYPE EL2809_2B6483BD EXTENDS TcoIo.EtcSlaveTerminalBase_947E5A46 :
STRUCT
	{attribute addProperty Name "Channel_1"}
	Channel_1 : Channel_42CA91F7;
	{attribute addProperty Name "Channel_2"}
	Channel_2 : Channel_42CA91F7;
	{attribute addProperty Name "Channel_3"}
	Channel_3 : Channel_42CA91F7;
	{attribute addProperty Name "Channel_4"}
	Channel_4 : Channel_42CA91F7;
	{attribute addProperty Name "Channel_5"}
	Channel_5 : Channel_42CA91F7;
	{attribute addProperty Name "Channel_6"}
	Channel_6 : Channel_42CA91F7;
	{attribute addProperty Name "Channel_7"}
	Channel_7 : Channel_42CA91F7;
	{attribute addProperty Name "Channel_8"}
	Channel_8 : Channel_42CA91F7;
	{attribute addProperty Name "Channel_9"}
	Channel_9 : Channel_42CA91F7;
	{attribute addProperty Name "Channel_10"}
	Channel_10 : Channel_42CA91F7;
	{attribute addProperty Name "Channel_11"}
	Channel_11 : Channel_42CA91F7;
	{attribute addProperty Name "Channel_12"}
	Channel_12 : Channel_42CA91F7;
	{attribute addProperty Name "Channel_13"}
	Channel_13 : Channel_42CA91F7;
	{attribute addProperty Name "Channel_14"}
	Channel_14 : Channel_42CA91F7;
	{attribute addProperty Name "Channel_15"}
	Channel_15 : Channel_42CA91F7;
	{attribute addProperty Name "Channel_16"}
	Channel_16 : Channel_42CA91F7;
	{attribute addProperty Name "WcState"}
	WcState : TcoIo.WcState_0B2B16F9;
	{attribute addProperty Name "InfoData"}
	InfoData : TcoIo.InfoData_6F19DB2B;
END_STRUCT
END_TYPE

// ---- DUTs/IO/Boxes/EL9011_D65D3D32.TcDUT
{attribute 'GeneratedUsingTerminal: EL9011--0000'}
{attribute addProperty VendorId "#x00000002"}
{attribute addProperty BoxType "EL9011--0000"}
{attribute addProperty Description "EL9011 End Terminal"}
{attribute addProperty Physics ""}
{attribute addProperty Id "EL9011"}
{attribute addProperty CRC "3596434738"}
{attribute addProperty Size "0"}
TYPE EL9011_D65D3D32 EXTENDS TcoIo.EtcSlaveEndTerminalBase_866C7F0C :
STRUCT
END_STRUCT
END_TYPE

// ---- DUTs/IO/Devices/SyncUnitTasks_4BE01469.TcDUT
{attribute 'GeneratedUsingTerminal: '}
{attribute addProperty BoxType ""}
{attribute addProperty Id "unreferencedAT %I*SyncUnitTask_AB2F50799PlcTaskAT %I*SyncUnitTask_AB2F50799"}
{attribute addProperty CRC "1272976489"}
{attribute addProperty Size "18"}
TYPE SyncUnitTasks_4BE01469 EXTENDS TcoIo.SyncUnitTasksBase_7C8711EB :
STRUCT
	{attribute addProperty Name "unreferenced"}
	unreferenced : TcoIo.SyncUnitTask_AB2F5079;
	{attribute addProperty Name "PlcTask"}
	PlcTask : TcoIo.SyncUnitTask_AB2F5079;
END_STRUCT
END_TYPE

// ---- DUTs/IO/Devices/SyncUnits_67D36DDA.TcDUT
{attribute 'GeneratedUsingTerminal: '}
{attribute addProperty BoxType ""}
{attribute addProperty Id "_defaultAT %I*SyncUnitTasks_4BE0146918"}
{attribute addProperty CRC "1741909466"}
{attribute addProperty Size "18"}
TYPE SyncUnits_67D36DDA EXTENDS TcoIo.SyncUnitsBase_AD6C35CE :
STRUCT
	{attribute addProperty Name "_default"}
	_default : SyncUnitTasks_4BE01469;
END_STRUCT
END_TYPE

// ---- DUTs/IO/Topology/EK_E812B8FA.TcDUT
{attribute 'GeneratedUsingTerminal: EK1122-0000-0018'}
{attribute addProperty BoxType "EK1122-0000-0018"}
{attribute addProperty Id "PNEUAES_510494FB88ABEPP1322_1FC0878B2AB21EPP1809_32157CFD20AB22EPP1809_32157CFD20AB23EPP1008_78E8D3DD12AB24EPP1008_78E8D3DD12"}
{attribute addProperty CRC "3893541114"}
{attribute addProperty Size "154"}
{attribute addProperty Name "EK"}
TYPE EK_E812B8FA EXTENDS EK1122_1FC0878B :
STRUCT
	{attribute addProperty Name "PNEU"}
	{attribute addProperty PreviousPort "EK : D"}
	{attribute addProperty SyncUnit "default"}
	PNEU : AES_510494FB;
	{attribute addProperty Name "AB"}
	{attribute addProperty PreviousPort "PNEU : B"}
	{attribute addProperty SyncUnit "default"}
	AB : EPP1322_1FC0878B;
	{attribute addProperty Name "AB21"}
	{attribute addProperty PreviousPort "AB : C"}
	{attribute addProperty SyncUnit "default"}
	AB21 : EPP1809_32157CFD;
	{attribute addProperty Name "AB22"}
	{attribute addProperty PreviousPort "AB21 : B"}
	{attribute addProperty SyncUnit "default"}
	AB22 : EPP1809_32157CFD;
	{attribute addProperty Name "AB23"}
	{attribute addProperty PreviousPort "AB22 : B"}
	{attribute addProperty SyncUnit "default"}
	AB23 : EPP1008_78E8D3DD;
	{attribute addProperty Name "AB24"}
	{attribute addProperty PreviousPort "AB23 : B"}
	{attribute addProperty SyncUnit "default"}
	AB24 : EPP1008_78E8D3DD;
END_STRUCT
END_TYPE

// ---- DUTs/IO/Topology/EC_4E5C738F.TcDUT
{attribute 'GeneratedUsingTerminal: EK1200-1388-0000'}
{attribute addProperty BoxType "EK1200-1388-0000"}
{attribute addProperty Id "EKEK_E812B8FA154IA1EL1809_32157CFD20QA1EL2809_2B6483BD19Term_11_EL9011EL9011_D65D3D320"}
{attribute addProperty CRC "1314681743"}
{attribute addProperty Size "193"}
{attribute addProperty Name "EC"}
TYPE EC_4E5C738F EXTENDS EK1200_013D0B49 :
STRUCT
	{attribute addProperty Name "EK"}
	{attribute addProperty PreviousPort "EC : B"}
	{attribute addProperty SyncUnit "default"}
	EK : EK_E812B8FA;
	{attribute addProperty Name "IA1"}
	{attribute addProperty PreviousPort "EK : C"}
	{attribute addProperty SyncUnit "default"}
	IA1 : EL1809_32157CFD;
	{attribute addProperty Name "QA1"}
	{attribute addProperty PreviousPort "IA1 : B"}
	{attribute addProperty SyncUnit "default"}
	QA1 : EL2809_2B6483BD;
	{attribute addProperty Name "Term 11 (EL9011)"}
	{attribute addProperty PreviousPort "QA1 : B"}
	{attribute addProperty SyncUnit "default"}
	Term_11_EL9011 : EL9011_D65D3D32;
END_STRUCT
END_TYPE

// ---- DUTs/IO/Topology/EC_245FBB9A.TcDUT
{attribute 'GeneratedUsingTerminal: IODEVICETYPE_ETHERCATPROT'}
{attribute addProperty BoxType "IODEVICETYPE_ETHERCATPROT"}
{attribute addProperty Id "ECEC_4E5C738F193SyncUnitsSyncUnits_67D36DDA18InputsInputs_A65FACA410OutputsOutputs_23C0ED1D6InfoDataInfoData_84133AC922"}
{attribute addProperty CRC "610253722"}
{attribute addProperty Size "249"}
{attribute addProperty Name "EC"}
TYPE EC_245FBB9A EXTENDS TcoIo.EtcMasterBase_62654B43 :
STRUCT
	{attribute addProperty Name "EC"}
	{attribute addProperty PreviousPort "EC : Master"}
	{attribute addProperty SyncUnit "default"}
	EC : EC_4E5C738F;
	{attribute addProperty Name "SyncUnits"}
	SyncUnits : SyncUnits_67D36DDA;
	{attribute addProperty Name "Inputs"}
	Inputs : TcoIo.Inputs_A65FACA4;
	{attribute addProperty Name "Outputs"}
	Outputs : TcoIo.Outputs_23C0ED1D;
	{attribute addProperty Name "InfoData"}
	InfoData : TcoIo.InfoData_84133AC9;
END_STRUCT
END_TYPE

// ---- GVLs/GVL_iXlinker.TcGVL
{attribute 'qualified_only'}
VAR_GLOBAL
		EC : EC_245FBB9A;
END_VAR

// ---- Abstractions/Components/MtsFeeding/TcoFeedingSequenceTask.TcPOU
FUNCTION_BLOCK TcoFeedingSequenceTask EXTENDS TcoCore.TcoTask
VAR
	_sequence      : TcoCore.TcoSequence(THIS^, eRestoreMode.None);
    _observerSequence       : TcoCore.TcoSequencerObserver(THIS^);
END_VAR

PROPERTY PUBLIC Observer : REFERENCE TO TcoCore.TcoSequencerObserver
GET
Observer ref=_observerSequence;
END_GET
END_PROPERTY

(*~
	<docu>
		<summary>
			Restores this instance to the Ready state. Can be called explicitly or from within one of the restore mechanisms.
			<para>
				See also <see cref="PlcDocu.TcoCore.TcoTask.AutoRestorable()"/>
			</para>
		</summary>			
	</docu>	
~*)
METHOD Restore : ITcoRestorable
SUPER^.Restore();
_sequence.Restore();
END_METHOD

PROPERTY PUBLIC Sequence : REFERENCE TO TcoCore.TcoSequence
GET
Sequence ref=_sequence;
END_GET
END_PROPERTY

END_FUNCTION_BLOCK

// ---- Abstractions/Components/MtsFeeding/TcoPlsPaletizator.TcPOU
FUNCTION_BLOCK TcoPlsPaletizator EXTENDS TcoCore.TcoComponent
VAR_INPUT
	inSafeCondition:BOOL;
	inDoorOpen:BOOL;
END_VAR

VAR_OUTPUT
END_VAR
VAR
	 {attribute addProperty Name "<#Config#>"}
	_config:TcoPlsPaletizator_Config_v_1_x_x;
	 {attribute addProperty Name "<#Status#>"}
    {attribute clr [ReadOnly()]}
	_status:TcoPlsPaletizator_Status_v_1_x_x;
	 {attribute addProperty Name "<#Control#>"}
	_control:TcoPlsPaletizator_Control_v_1_x_x;
	
	 {attribute addProperty Name "<#Components#>"}
    _components:TcoPlsPaletizator_Components:= (Parent := THIS^);
	
	{attribute addProperty Name "<#Poziadavka novy blister#>"}
	_feedNewBlisterTask : TcoFeedingSequenceTask(THIS^);
	{attribute addProperty Name "<#Poziadavka vylozenie blistera#>"}
	_throwBlisterTask :  TcoFeedingSequenceTask(THIS^);
	{attribute addProperty Name "<#Poziadavka obsluhy vystupny buffer#>"}
	_hanldeOutBufferTask :  TcoFeedingSequenceTask(THIS^);


	
	{attribute addProperty Name "<#Restore#>"}
	_restoreTask:TcoCore.TcoTask(THIS^);

	_blinker:TcoBlinker(THIS^);
	restoreDone: BOOL;
END_VAR

_status.SafeCondition:=inSafeCondition;
_status.EntryBufferEmpty:=NOT Components.I3_PresentBlistersInBufferEmpty.Signal;
_status.BlisterReady:= Components.I4_PresentBlisterInWorkingPos.Signal ;
_status.OutBufferFull:= Components.I8_OutBlistersBufferIsFull.Signal;

_feedNewBlisterTask.Enabled :=NOT _throwBlisterTask.Busy;
IF(_feedNewBlisterTask.Execute())THEN
	SequenceIncomingBlister(refSequenceTask:=_feedNewBlisterTask );
END_IF;

_throwBlisterTask.Enabled :=NOT _feedNewBlisterTask.Busy;
IF(_throwBlisterTask.Execute())THEN
	SequenceOutgoingBlister(refSequenceTask:=_throwBlisterTask);
END_IF;

_hanldeOutBufferTask.Enabled :=TRUE;
IF(_hanldeOutBufferTask.Execute())THEN
	SequenceOutgoingBuffer(refSequenceTask:=_hanldeOutBufferTask);
END_IF;



//*************RESTORE********************

_restoreTask.Enabled := TRUE;
IF _restoreTask.Execute() THEN
	Restore();
	restoreDone:= Components.P3_HorizontalSepareEntryBlisters.MoveToWork().Done AND (Components.P10_HoldEntrySepareOutBlister.MoveToHome().Done or _config.SepareBlistersAtEntryInactive)
		AND_THEN (Components.P1_VerticalSepareEntryBlisters.MoveToHome().Done AND Components.P2_VerticalSepareEntryBlisters.MoveToHome().Done)
		AND_THEN (Components.P5_HorizontalSepareOutBlisters.MoveToHome().Done AND_THEN Components.P6_VerticalSepareOutBlister.MoveToHome().Done)
		AND_THEN  Components.P4_FeedEntryBlister.MoveToHome().Done;
		
	
	_restoreTask.DoneWhen(restoreDone);
END_IF
//****************************************

PROPERTY Components : REFERENCE TO TcoPlsPaletizator_Components
GET
Components ref=_components;
END_GET
END_PROPERTY

(*~
	<docu>
		<summary>
			Gets the configuration of the MTS Pls feeder. 					
		</summary>			
	</docu>	
~*)
PROPERTY Config : REFERENCE TO TcoPlsPaletizator_Config_v_1_x_x
GET
Config REF= _config;
END_GET
END_PROPERTY

METHOD PUBLIC DefaultSignalisation
VAR_INPUT
END_VAR
Components.Q1_AttentionSignalisationR.Reset();
Components.Q2_AttentionSignalisationG.Reset();
Components.Q3_AttentionSignalisationB.Reset();

_blinker(inOffTime:=_config.BlinkTime,inOnTime:=_config.BlinkTime);

IF NOT _status.OutBufferFull 
	AND NOT _status.EntryBufferEmpty THEN
	Components.Q2_AttentionSignalisationG.Set();
ELSIF  _blinker.IsOn THEN
	IF inDoorOpen AND 
		THIS^._feedNewBlisterTask.Busy
		OR
		THIS^._throwBlisterTask.Busy
		OR
		THIS^._hanldeOutBufferTask.Busy THEN
		Messenger.Warning('<#CAKANIE NA OBSLUHU PALETIZERA - ZAVRITE DVERE!#>');
		Components.Q1_AttentionSignalisationR.Set();
		Components.Q2_AttentionSignalisationG.Set();
	ELSIF NOT _status.OutBufferFull
		AND _status.EntryBufferEmpty
		AND _status.BlisterReady THEN
		
		Components.Q1_AttentionSignalisationR.Set();
		Components.Q2_AttentionSignalisationG.Set();

	ELSIF NOT _status.OutBufferFull
		AND _status.EntryBufferEmpty 
		AND NOT _status.BlisterReady THEN	
		Components.Q1_AttentionSignalisationR.Set();
	ELSIF  _status.OutBufferFull  THEN
		Components.Q1_AttentionSignalisationR.Set();	
	
	END_IF;


	
END_IF;
END_METHOD

PROPERTY FeedNewBlisterTask : REFERENCE TO TcoFeedingSequenceTask
GET
FeedNewBlisterTask ref=_feedNewBlisterTask;
END_GET
END_PROPERTY

PROPERTY HandleOutBufferTask : REFERENCE TO TcoFeedingSequenceTask
GET
HandleOutBufferTask ref=_hanldeOutBufferTask;
END_GET
END_PROPERTY

(*~
	<docu>
		<summary>
			Restores this instance to the Ready state. Can be called explicitly or from within one of the restore mechanisms.	
		</summary>			
	</docu>	
~*)
METHOD  Restore : ITcoRestorable

_hanldeOutBufferTask.Restore();
_feedNewBlisterTask.Restore();
_throwBlisterTask.Restore();
END_METHOD

METHOD PUBLIC SafetyBlockingMovements
VAR_INPUT
END_VAR
//********************SAFETY******************

Components.P4_FeedEntryBlister.SuspendMoveWorkExpression(NOT Components.P7_SupportEntryBlister.AtHome ,'Movement is blocked due P7 is not in home position');
Components.P4_FeedEntryBlister.SuspendMoveHomeExpression(NOT Components.P6_VerticalSepareOutBlister.AtHome,'Movement is blocked due P6 is not in home position');
END_METHOD

METHOD SequenceIncomingBlister
VAR_INPUT
	refSequenceTask : REFERENCE TO TcoFeedingSequenceTask;
	
	
END_VAR

VAR
    seq    : REFERENCE TO TcoCore.TcoSequence;


END_VAR
seq REF= refSequenceTask.Sequence;

seq.Open();
seq.Observer := refSequenceTask.Observer;



		



//***************************************************************************************************     
//    This step will be executed and immediately finished, as the condition in Await method is true.
IF seq.Step(0,TRUE,'<#INIT#>') THEN   
	Messenger.Warning('<#BEZPECNOST ZARIADENIA NARUSENA. NIEJE MOZNE VYKONAT AKCIU#>');     
	IF _status.SafeCondition THEN
    	seq.CompleteStep();
	END_IF;
END_IF        
//***************************************************************************************************     

 
//***************************************************************************************************     
IF seq.Step(10,TRUE,'<#KONTROLA POCTU VSTUPNYCH BLISTROV#>') THEN   
    Messenger.Warning('<#PODAVAC PRAZDNY! DOPLNE VSTUPNE BLISTRE !#>');
    seq.StepCompleteWhen(Components.I3_PresentBlistersInBufferEmpty.IsTrue);
END_IF        
//***************************************************************************************************     


        
//***************************************************************************************************     
IF seq.Step(20,TRUE,'<#SEPAROVANIE VSTUPNEHO BLISTRA - VERTIKALNE VALCE VYSUNUTE#>') THEN   

    seq.StepCompleteWhen(THIS^.Components.P1_VerticalSepareEntryBlisters.MoveToWork().Done AND THIS^.Components.P2_VerticalSepareEntryBlisters.MoveToWork().Done);
END_IF        
//***************************************************************************************************     


//***************************************************************************************************     
IF seq.Step(30,TRUE,'<#SEPAROVANIE VSTUPNEHO BLISTRA - SEPAROVANIE ZASUNUTE#>') THEN   

    seq.StepCompleteWhen(THIS^.Components.P3_HorizontalSepareEntryBlisters.MoveToHome().Done);
END_IF        
//***************************************************************************************************     


//***************************************************************************************************     
IF seq.Step(40,TRUE,'<#SEPAROVANIE VSTUPNEHO BLISTRA - VERTIKALNE VALCE ZASUNUT JEDEN#>') THEN   

    seq.StepCompleteWhen(THIS^.Components.P1_VerticalSepareEntryBlisters.MoveToHome().Done AND_THEN THIS^.Components.P2_VerticalSepareEntryBlisters.MoveToWork().Done);
END_IF        
//***************************************************************************************************     


//***************************************************************************************************     
IF seq.Step(50,TRUE,'<#SEPAROVANIE VSTUPNEHO BLISTRA - SEPAROVANIE VYSUNUTE#>') THEN   

    seq.StepCompleteWhen(THIS^.Components.P3_HorizontalSepareEntryBlisters.MoveToWork().Done AND (Components.P10_HoldEntrySepareOutBlister.MoveToWork().Done or _config.SepareBlistersAtEntryInactive));
END_IF        
//***************************************************************************************************     

//***************************************************************************************************     
IF seq.Step(60,TRUE,'<#SEPAROVANIE VSTUPNEHO BLISTRA - VERTIKALNE VALCE ZASUNUT OBIDVA#>') THEN   

    seq.StepCompleteWhen(THIS^.Components.P1_VerticalSepareEntryBlisters.MoveToHome().Done AND THIS^.Components.P2_VerticalSepareEntryBlisters.MoveToHome().Done 
						AND_THEN (Components.P10_HoldEntrySepareOutBlister.MoveToHome().Done) OR _config.SepareBlistersAtEntryInactive);
END_IF        
//***************************************************************************************************     

//***************************************************************************************************   
IF seq.Step(70,TRUE,'<#KONTROLA PRITOMNOSTI SEPAROVANEHO KUSU#>') THEN   
    Messenger.Error('<#PODAVAC PRAZDNY! DOPLNE BLISTRE !#>');
    seq.StepCompleteWhen(THIS^.Components.I1_PresentBlisterEntry.IsTrue AND (THIS^.Components.I2_PresentBlisterEntryEmptySpace.IsTrue) );
END_IF        
//***************************************************************************************************     


//***************************************************************************************************     
IF seq.Step(80,TRUE,'<#SEPAROVANIE VSTUPNEHO BLISTRA - PRESUNUTIE BLISTRA DO POZICIE ODOBERANIA#>') THEN   

    seq.StepCompleteWhen(THIS^.Components.P8_FixEntryBlisterSide.MoveToHome().Done AND_THEN THIS^.Components.P4_FeedEntryBlister.MoveToWork().Done AND Components.i4_PresentBlisterInWorkingPos.IsTrue);
END_IF        
//***************************************************************************************************     


//***************************************************************************************************     
IF seq.Step(90,TRUE,'<#SEPAROVANIE VSTUPNEHO BLISTRA - UPEVENIE BLISTRA ZBOKU#>') THEN   

    seq.StepCompleteWhen(THIS^.Components.P8_FixEntryBlisterSide.MoveToWork().Done);
END_IF        
//***************************************************************************************************     



//***************************************************************************************************     
IF seq.Step(100,TRUE,'<#SEPAROVANIE VSTUPNEHO BLISTRA - NPRESUNUTIE BLISTRA DO POZICIE NABERANIA#>') THEN   

   IF THIS^.Components.P6_VerticalSepareOutBlister.AtHome THEN
	    seq.CompleteStep();
	ELSE
		Messenger.Error('VYSTUPNY BUFFER NIEJE V HORNEJ POZICII!(P6)');
	END_IF
END_IF        
//***************************************************************************************************   

//***************************************************************************************************     
IF seq.Step(110,TRUE,'<#SEPAROVANIE VSTUPNEHO BLISTRA - ZASUNUTE P4#>') THEN   

	 seq.StepCompleteWhen(THIS^.Components.P4_FeedEntryBlister.MoveToHome().Done) ;
	
END_IF        
//***************************************************************************************************   


//***************************************************************************************************     
IF seq.Step(120,TRUE,'SEPAROVANIE VSTUPNEHO BLISTRA - NPRESUNUTIE BLISTRA DO POZICIE NABERANIA') THEN   

    seq.StepCompleteWhen(THIS^.Components.P7_SupportEntryBlister.MoveToWork().Done AND (THIS^.Components.P9_LockEntryBlisterTop.MoveToHome().Done OR _config.LockBlisterInPickPosInactive));
END_IF        
//***************************************************************************************************   




IF (seq.Step(inStepID := seq.RESTORE_STEP_ID,
    inEnabled := TRUE,
    inStepDescription := 'RETURN TO THE START OF THE SEQUENCE')) THEN
    //--------------------------------------------------------	
		refSequenceTask.DoneWhen(TRUE);
    	seq.CompleteSequence();
    //--------------------------------------------------------			
END_IF;

seq.Close();
END_METHOD

METHOD SequenceOutgoingBlister
VAR_INPUT
	refSequenceTask : REFERENCE TO TcoFeedingSequenceTask;
	
	
END_VAR

VAR
    seq    : REFERENCE TO TcoCore.TcoSequence;

END_VAR

VAR_INST
	_timer:ton;
	
END_VAR
seq REF= refSequenceTask.Sequence;

seq.Open();
seq.Observer := refSequenceTask.Observer;



		



//***************************************************************************************************     
//    This step will be executed and immediately finished, as the condition in Await method is true.
IF seq.Step(0,TRUE,'<#INIT#>') THEN   
	Messenger.Warning('<#BEZPECNOST ZARIADENIA NARUSENA. NIEJE MOZNE VYKONAT AKCIU#>');     
	IF _status.SafeCondition THEN
    	seq.CompleteStep();
	END_IF;
END_IF        
//***************************************************************************************************     

IF seq.Step(10,TRUE,'<#SEPAROVANIE VYSTUPNEHO BLISTRA - UVOLNENIE BLISTRA#>') THEN   

    seq.StepCompleteWhen( (THIS^.Components.P9_LockEntryBlisterTop.MoveToWork().Done OR _config.LockBlisterInPickPosInactive) AND THIS^.Components.P8_FixEntryBlisterSide.MoveToHome().Done);
END_IF        
//***************************************************************************************************   


//***************************************************************************************************     
IF seq.Step(20,TRUE,'<#SEPAROVANIE VYSTUPNEHO BLISTRA - ZASUNUTIE SUPPORTU#>') THEN   

   seq.StepCompleteWhen(THIS^.Components.P7_SupportEntryBlister.MoveToHome().Done);
END_IF        
//***************************************************************************************************   



//***************************************************************************************************     
IF seq.Step(30,TRUE,'<#SEPAROVANIE VYSTUPNEHO BLISTRA - KONTROLA PRITOMNOSTI BLISTA NA SKLZE#>') THEN   
	IF seq.IsFreshState THEN
		_timer(IN:=FALSE);
	END_IF
	_timer(IN:=THIS^.Components.I5_OutBlistersIsThrowedCorrectly.Signal,PT:=_config.StabilisationTime);
	
    seq.StepCompleteWhen(_timer.Q);
END_IF        
//***************************************************************************************************   



IF (seq.Step(inStepID := seq.RESTORE_STEP_ID,
    inEnabled := TRUE,
    inStepDescription := 'RETURN TO THE START OF THE SEQUENCE')) THEN
    //--------------------------------------------------------	
		refSequenceTask.DoneWhen(TRUE);
    	seq.CompleteSequence();
    //--------------------------------------------------------			
END_IF;

seq.Close();
END_METHOD

METHOD SequenceOutgoingBuffer
VAR_INPUT
	refSequenceTask : REFERENCE TO TcoFeedingSequenceTask;
	
	
END_VAR

VAR
    seq    : REFERENCE TO TcoCore.TcoSequence;

END_VAR

VAR_INST
	_timer:ton;
	
END_VAR
seq REF= refSequenceTask.Sequence;

seq.Open();
seq.Observer := refSequenceTask.Observer;



		



//***************************************************************************************************     
//    This step will be executed and immediately finished, as the condition in Await method is true.
IF seq.Step(0,TRUE,'<#INIT#>') THEN   
	Messenger.Warning('<#BEZPECNOST ZARIADENIA NARUSENA. NIEJE MOZNE VYKONAT AKCIU#>');     
	IF _status.SafeCondition THEN
    	seq.CompleteStep();
	END_IF;
END_IF        
//***************************************************************************************************     



//***************************************************************************************************     
IF seq.Step(10,TRUE,'<#VYSTUPNY BUFFER - KONTROLA PRITOMNOSTI BLISTA NAD BUFFEROM#>') THEN   
	IF seq.IsFreshState THEN
		_timer(IN:=FALSE);
	END_IF
	_timer(IN:=NOT THIS^.Components.I5_OutBlistersIsThrowedCorrectly.Signal AND Components.I7_OutBlistersIsAboveOutBuffer.Signal,PT:=_config.StabilisationTime);
	
    seq.StepCompleteWhen(_timer.Q);
END_IF        
//***************************************************************************************************   


//***************************************************************************************************     
IF seq.Step(20,TRUE,'<#VYSTUPNY BUFFER - KONTROLA POSCTU BLISTROV#>') THEN   
	Messenger.Error('<#PODAVAC PLNY! ODSTRANTE PRAZDNE BLISTRE !#>');
    seq.StepCompleteWhen(THIS^.Components.I8_OutBlistersBufferIsFull.IsFalse);
END_IF        
//***************************************************************************************************   


//***************************************************************************************************     
IF seq.Step(30,TRUE,'<#VYSTUPNY BUFFER - POSUN KUSOV NAD BUFFER#>') THEN   

	THIS^.Components.P6_VerticalSepareOutBlister.MoveToWork();
	IF Components.I6_OutBlistersLisftSignal.Signal THEN
	
		THIS^.Components.P6_VerticalSepareOutBlister.MoveWorkTask.Abort();
	    seq.StepCompleteWhen(TRUE);
	END_IF;
		
END_IF        
//***************************************************************************************************   


//***************************************************************************************************     
IF seq.Step(40,TRUE,'<#VYSTUPNY BUFFER - UVOLNENIE BLISTRA A NAVRAT NAHOR#>') THEN   

	
	seq.StepCompleteWhen(Components.P5_HorizontalSepareOutBlisters.MoveToWork().Done AND_THEN THIS^.Components.P6_VerticalSepareOutBlister.MoveToHome().Done);
		
END_IF        
//***************************************************************************************************   

//***************************************************************************************************     
IF seq.Step(50,TRUE,'<#VYSTUPNY BUFFER - HORIZONTALNE ZASUNUTIE#>') THEN   

	
	seq.StepCompleteWhen(Components.P5_HorizontalSepareOutBlisters.MoveToHome().Done);
		
END_IF        
//***************************************************************************************************   



IF (seq.Step(inStepID := seq.RESTORE_STEP_ID,
    inEnabled := TRUE,
    inStepDescription := 'RETURN TO THE START OF THE SEQUENCE')) THEN
    //--------------------------------------------------------	
		refSequenceTask.DoneWhen(TRUE);
    	seq.CompleteSequence();
    //--------------------------------------------------------			
END_IF;

seq.Close();
END_METHOD

(*~
	<docu>
		<summary>
		    Custom service (manual, maintenance) logic.
			This method must be implemented in derived class.
		</summary>			
	</docu>	
~*)
METHOD PROTECTED  ServiceMode
_components.Q3_AttentionSignalisationB.Service();
_components.Q2_AttentionSignalisationG.Service();
_components.Q1_AttentionSignalisationR.Service();
_components.P1_VerticalSepareEntryBlisters.Service();
_components.P2_VerticalSepareEntryBlisters.Service();
_components.P3_HorizontalSepareEntryBlisters.Service();
_components.P4_FeedEntryBlister.Service();
_components.P5_HorizontalSepareOutBlisters.Service();
_components.P6_VerticalSepareOutBlister.Service();
_components.P7_SupportEntryBlister.Service();
_components.P8_FixEntryBlisterSide.Service();
_components.P9_LockEntryBlisterTop.Service();
_components.P10_HoldEntrySepareOutBlister.Service();
END_METHOD

(*~
	<docu>
		<summary>
			Gets the status of the MTS Pls feeder. 					
		</summary>			
	</docu>	
~*)
PROPERTY Status : REFERENCE TO TcoPlsPaletizator_Status_v_1_x_x
GET
Status REF= _status;
END_GET
END_PROPERTY

PROPERTY ThrowBlisterTask : REFERENCE TO TcoFeedingSequenceTask
GET
ThrowBlisterTask ref=_throwBlisterTask;
END_GET
END_PROPERTY

END_FUNCTION_BLOCK

// ---- Technology/CU00x/Safety/Suspend/CU00xSuspendTask.TcPOU
FUNCTION_BLOCK CU00xSuspendTask EXTENDS CUBaseSuspend IMPLEMENTS ICUTask
VAR

	
	
	_sb : TcoCore.StringBuilder;
END_VAR

VAR

END_VAR

Run();

(*~
	<docu>
		<summary>
			Main method of the sequener. Custom code needs to be placed here. The sequencer is executed by call of **Instance.Run()** method.
			This method is abstract, and it must be overridden in derived block.
		</summary>
	</docu>
~*)
METHOD PROTECTED Main : BOOL
(*

	SUSPEND PROCESS 
	Following steps provide suspend actions for this controlled unit.
	Add components add write customized sequence according to your need.
*)

		
//
IF (Step(100, TRUE, '<#WAITING FOR START#>')) THEN
    //-------------------------------------    

    StepCompleteWhen(TRUE);
    //-------------------------------------
END_IF

//HERE  YOU CAN WRITE  WHAT IS NECESSARY 
//TO SUPSEND  PROCESS..... TO INTERUPT SAFETY

IF (Step(1000, TRUE, '<#SUSPENDING COMPONENTS#>')) THEN
 	//-------------------------------------    
	//StepCompleteWhen(Station.AutomatTask.CurrentStep.Status <> eStepStatus.Running);
		
    StepCompleteWhen( CurrentStep.Duration >= T#3000MS);
    //-------------------------------------
END_IF

IF (Step(30000, TRUE, 'SUSPEND DONE')) THEN
    //-------------------------------------
		
        THIS^._done:=TRUE;
		THIS^.Task.DoneWhen(TRUE);
	
   
    //-------------------------------------	
END_IF
END_METHOD

METHOD PUBLIC OnStart
SUPER^.OnStart();
Station.RecoverTask.Restore();
END_METHOD

PROPERTY Station : REFERENCE TO CU00x
GET
VAR
    _station : POINTER TO CU00x;
END_VAR
IF __QUERYPOINTER(Parent, _station) THEN // Check if _Parent is Station001
    Station REF= _station^;              // If the check is successful dereference a pointer. simlar to THIS^ or SUPER^
END_IF
END_GET
END_PROPERTY

END_FUNCTION_BLOCK

// ---- Technology/CU00x/CU00x.TcPOU
{attribute addProperty ShortName "CU00x"}
{attribute addProperty Name "Controlled unit x_tempalte_x"}
FUNCTION_BLOCK CU00x EXTENDS CUBase 
VAR
    _cuProcessDataDisplay       :  CU00xProcessData := (Parent := THIS^);
    _cuTechnologicalDataDisplay :  CU00xTechnologicalData := (Parent := THIS^);
    _components          		:  CU00xComponents := (Parent := THIS^);
	{attribute addProperty Name "<#MANUAL#>"}
    {attribute addProperty ToolTip "<#Start manual/Service mode#>"}	
    _manualTask : CU00xManualTask(THIS^);
	{attribute addProperty Name "<#GROUND#>"}
    {attribute addProperty ToolTip "<#Brings the device into basic position.#>"}
    _groundTask : CU00xGroundTask(THIS^, TcoCore.eRestoreMode.None);
    {attribute addProperty Name "<#AUTOMAT#>"}
    {attribute addProperty ToolTip "<#Starts automatic sequence. Before start you need to perform grounding sequence.#>"}	
    _automatTask : CU00xAutomatTask(THIS^, TcoCore.eRestoreMode.None);     
	
	 {attribute addProperty Name "<#SUSPEND PROCESS#>"}
    {attribute addProperty ToolTip "<#Starts suspend sequence of process(automatic,ground sequence). #>"}	
    _suspendTask : CU00xSuspendTask(THIS^, TcoCore.eRestoreMode.None);     
	
	{attribute addProperty Name "<#RECOVER PROCESS#>"}
    {attribute addProperty ToolTip "<#Starts suspend sequence of process(automatic,ground sequence). #>"}	
    _recoverTask : CU00xRecoverTask(THIS^, TcoCore.eRestoreMode.None);     
  	
	{attribute addProperty Name "<#Test positions#>"}
	_positions : Cu00xTestPositions(THIS^);


	{attribute addProperty Name "<#Test multi positions#>"}
	 _positionsMulti : CU00xTestMultiPositions(THIS^);

END_VAR

THIS^.CuId := eStations.CU00x;



(*
	This controlled unit's component initialization.
*)

THIS^.InitializeComponents();

(*
	This controlled unit process data crud operations handler.
	Control exchange of process data between this controlled unit and the data repository.
*)

_processData();
_productionPlaner();


(*
	
	Cu's Modes
	
*)

Automat();
Ground();
Manual();


_suspendTask();
_recoverTask();







(*
	When no mode is active 'Idle' method should be called.
	'NoMode' method shouls contain code that renders this cu idle. 
*)

IF NOT (AutomatTask.Task.Busy 
		OR GroundTask.Task.Busy
		OR ManualTask.Task.Busy) 
THEN
	Idle();
END_IF



(*
	Updates this controlled unit's information for the UI.
*)


UpdateInfo();

_cuProcessDataDisplay := ProcessDataManager.Data.CU00x;
_cuTechnologicalDataDisplay := Technology.TechnologicalSettings.Data.CU00x;

_settings.WarningCycleTime:= _cuTechnologicalDataDisplay.WarningCycleTime;
_settings.ErrorCycleTime:= _cuTechnologicalDataDisplay.ErrorCycleTime;
_settings.AnyRecurringFailure:= _cuTechnologicalDataDisplay.AnyRecurringFailure;
_settings.SameRecurringFailure:= _cuTechnologicalDataDisplay.SameRecurringFailure;

(*~
	<docu>
		<summary>
			Controls `automatic` mode of `CU00x`.
		</summary>
	</docu>
~*)
METHOD Automat
VAR_INPUT
END_VAR
(*
	Enable condition to start `automatTask`.
	Modify according your needs.
	[! 
	THIS IS NOT SAFETY CONDITION. THE SAFETY OF PRESONNEL AND EQUIPMENT MUST BE ENSURED BY ADDITIONAL MEANS 
	TO COMPLY WITH REGULATIONS
	]
*)


//_automatTask.Task.Enabled := (_groundTask.GroundDone OR  _automatTask.Task.Busy) AND THIS^.Technology.AllowAutomat();

(*
	Invokes `groundTask` from technology object.
*)

//IF(Technology.AutomatAllTask.Execute()) THEN _automatTask.Task.Invoke(); END_IF;

//IF(Technology.ForceStepMode()) THEN
 //	_automatTask.ModeController.Mode := eSequencerMode.StepMode;
//END_IF 



(*
	or use default behavior from abstraction
*)
	SUPER^.Automat();

(*

	Executes sequence of automatic mode.

*)

_automatTask();
END_METHOD

PROPERTY AutomatTask : REFERENCE TO CUBaseAutomat
GET
AutomatTask REF= _automatTask;
END_GET
END_PROPERTY

PROPERTY Components : REFERENCE TO CU00xComponents
GET
Components REF= _components;
END_GET
END_PROPERTY

(*~
	<docu>
		<summary>
			Controls `ground` mode of `CU00x`.
		</summary>
	</docu>
~*)
METHOD Ground : BOOL
VAR_INPUT
END_VAR
(*
	Enable condition to start `groundTask`.
	Modify according your needs.
	[! 
	THIS IS NOT SAFETY CONDITION. THE SAFETY OF PRESONNEL AND EQUIPMENT MUST BE ENSURED BY ADDITIONAL MEANS 
	TO COMPLY WITH REGULATIONS
	]
*)

//_groundTask.Task.Enabled :=  THIS^.Technology.AllowGround();

(*
	Invokes `groundTask` from technology object.
*)

//IF(Technology.GroundAllTask.Execute()) THEN _groundTask.Task.Invoke(); END_IF;


//IF _groundTask.GroundDone AND _groundTask.Task.Execute() THEN _groundTask.Restore();_groundTask.Task.Invoke();END_IF;


(*
	or use default behavior from abstraction
*)
	SUPER^.Ground();




(*

	Executes sequence of groundTask.

*)

_groundTask();
END_METHOD

PROPERTY GroundTask : REFERENCE TO CUBaseGround
GET
GroundTask REF= _groundTask;
END_GET
END_PROPERTY

(*~
	<docu>
		<summary>
			Code to be called cylically when `CU00x` idle; no other mode is active.
		</summary>
	</docu>
~*)
METHOD Idle : BOOL
END_METHOD

METHOD InitializeComponents : BOOL

VAR_INST
	tempBoolHome: BOOL;
	tempBoolWork: BOOL;
	tempBoolP4Home: BOOL;
	tempBoolP4Work: BOOL;
END_VAR

Components.PairTagTask();
(*
components.Group1.horizontalCylinder(inoAtHomePos:=GVL_iXlinker.EC1.EK1200.IA1_EL1809.Channel_1.Input, 
							   inoAtWorkPos:=GVL_iXlinker.EC1.EK1200.IA1_EL1809.Channel_2.Input, 
							   inoToHomePos:=GVL_iXlinker.EC1.EK1200.IA1_EL1809.Channel_3.Input, 
							   inoToWorkPos:=GVL_iXlinker.EC1.EK1200.IA1_EL1809.Channel_4.Input);
Components.SingleAxis.Config.InfoTime:=T#4S;
Components.SingleAxis.Config.ErrorTime:=T#10S;



Components.SingleAxis(inEnable := ,
    inEnablePositive := ,
    inEnableNegative := ,
    inCalibrationCam := ,
    refAxis := GVL_iXlinker.Axis1,
	inoPositions:= _positions);
	
	

//Components.PickAndPlace();
//Components.PickAndPlace.Service();
		
Components.MultiAxis(inEnableAxis1 := ,
    inEnablePositiveAxis1 := ,
    inEnableNegativeAxis1 := ,
    inCalibrationCamAxis1 := ,
    refAxis1 := GVL_iXlinker.Axis1,
	inoPositions:= _positionsMulti);
	
			
//Components.PickAndPlace.Components.Manipulator(inEnableAxis1 := ,
//    inEnablePositiveAxis1 := ,
//    inEnableNegativeAxis1 := ,
//    inCalibrationCamAxis1 := ,
//    refAxis1 := GVL_iXlinker.Axis1,
//	inoPositions:= _positionsMulti);
*)

Components.PlsPaletizator.Components.I1_PresentBlisterEntry(inoSignal:=GVL_iXlinker.Ec.EC.EK.AB23.Channel_1.Input);
Components.PlsPaletizator.Components.I2_PresentBlisterEntryEmptySpace(inoSignal:=GVL_iXlinker.Ec.EC.Ek.AB23.Channel_2.Input);
Components.PlsPaletizator.Components.I3_PresentBlistersInBufferEmpty(inoSignal:=GVL_iXlinker.Ec.EC.Ek.AB23.Channel_3.Input);
Components.PlsPaletizator.Components.I4_PresentBlisterInWorkingPos(inoSignal:=GVL_iXlinker.Ec.EC.Ek.AB23.Channel_4.Input);
Components.PlsPaletizator.Components.I5_OutBlistersIsThrowedCorrectly(inoSignal:=GVL_iXlinker.Ec.EC.Ek.AB23.Channel_5.Input);
Components.PlsPaletizator.Components.I6_OutBlistersLisftSignal(inoSignal:=GVL_iXlinker.Ec.EC.Ek.AB23.Channel_6.Input);
Components.PlsPaletizator.Components.I7_OutBlistersIsAboveOutBuffer(inoSignal:=GVL_iXlinker.Ec.EC.Ek.AB23.Channel_7.Input);
Components.PlsPaletizator.Components.I8_OutBlistersBufferIsFull(inoSignal:=GVL_iXlinker.Ec.EC.Ek.AB23.Channel_8.Input);



Components.PlsPaletizator.Components.P1_VerticalSepareEntryBlisters
				(inoAtHomePos:=GVL_iXlinker.Ec.EC.Ek.AB21.Channel_1.Input,
				inoAtWorkPos:=GVL_iXlinker.Ec.EC.Ek.AB21.Channel_2.Input,
				inoToHomePos:=tempBoolHome,
				inoToWorkPos:=tempBoolWork);
GVL_iXlinker.Ec.EC.Ek.PNEU.Modules.Outputs.digital_Data_O[0].1:=tempBoolHome;
GVL_iXlinker.Ec.EC.Ek.PNEU.Modules.Outputs.digital_Data_O[0].0:=tempBoolWork;

Components.PlsPaletizator.Components.P2_VerticalSepareEntryBlisters
				(inoAtHomePos:=GVL_iXlinker.Ec.EC.Ek.AB21.Channel_3.Input,
				inoAtWorkPos:=GVL_iXlinker.Ec.EC.Ek.AB21.Channel_4.Input,
				inoToHomePos:=tempBoolHome,
				inoToWorkPos:=tempBoolWork);
GVL_iXlinker.Ec.EC.Ek.PNEU.Modules.Outputs.digital_Data_O[0].3:=tempBoolHome;
GVL_iXlinker.Ec.EC.Ek.PNEU.Modules.Outputs.digital_Data_O[0].2:=tempBoolWork;


Components.PlsPaletizator.Components.P3_HorizontalSepareEntryBlisters
				(inoAtHomePos1:=GVL_iXlinker.Ec.EC.Ek.AB21.Channel_5.Input,
				inoAtWorkPos1:=GVL_iXlinker.Ec.EC.Ek.AB21.Channel_6.Input,
				inoAtHomePos2:=GVL_iXlinker.Ec.EC.Ek.AB21.Channel_7.Input,
				inoAtWorkPos2:=GVL_iXlinker.Ec.EC.Ek.AB21.Channel_8.Input,
				inoToHomePos:=tempBoolHome,
				inoToWorkPos:=tempBoolWork);
GVL_iXlinker.Ec.EC.Ek.PNEU.Modules.Outputs.digital_Data_O[0].5:=tempBoolHome;
GVL_iXlinker.Ec.EC.Ek.PNEU.Modules.Outputs.digital_Data_O[0].4:=tempBoolWork;

Components.PlsPaletizator.Components.P4_FeedEntryBlister
				(inoAtHomePos:=GVL_iXlinker.Ec.EC.Ek.AB21.Channel_9.Input,
				inoAtWorkPos:=GVL_iXlinker.Ec.EC.Ek.AB21.Channel_10.Input,
				inoToHomePos:=tempBoolP4Home,
				inoToWorkPos:=tempBoolP4Work);
				Components.PlsPaletizator.SafetyBlockingMovements();

GVL_iXlinker.Ec.EC.Ek.PNEU.Modules.Outputs.digital_Data_O[0].7:=tempBoolP4Home;
GVL_iXlinker.Ec.EC.Ek.PNEU.Modules.Outputs.digital_Data_O[0].6:=tempBoolP4Work;

Components.PlsPaletizator.Components.P5_HorizontalSepareOutBlisters
				(inoAtHomePos1:=GVL_iXlinker.Ec.EC.Ek.AB21.Channel_11.Input,
				inoAtWorkPos1:=GVL_iXlinker.Ec.EC.Ek.AB21.Channel_12.Input,
				inoAtHomePos2:=GVL_iXlinker.Ec.EC.Ek.AB21.Channel_13.Input,
				inoAtWorkPos2:=GVL_iXlinker.Ec.EC.Ek.AB21.Channel_14.Input,
				inoToHomePos:=tempBoolHome,
				inoToWorkPos:=tempBoolWork);
GVL_iXlinker.Ec.EC.Ek.PNEU.Modules.Outputs.digital_Data_O[1].1:=tempBoolHome;
GVL_iXlinker.Ec.EC.Ek.PNEU.Modules.Outputs.digital_Data_O[1].0:=tempBoolWork;

Components.PlsPaletizator.Components.P6_VerticalSepareOutBlister
				(inoAtHomePos:=GVL_iXlinker.Ec.EC.Ek.AB21.Channel_15.Input,
				inoAtWorkPos:=GVL_iXlinker.Ec.EC.Ek.AB21.Channel_16.Input,
				inoToHomePos:=tempBoolHome,
				inoToWorkPos:=tempBoolWork);
GVL_iXlinker.Ec.EC.Ek.PNEU.Modules.Outputs.digital_Data_O[1].3:=tempBoolHome;
GVL_iXlinker.Ec.EC.Ek.PNEU.Modules.Outputs.digital_Data_O[1].2:=tempBoolWork;


Components.PlsPaletizator.Components.P7_SupportEntryBlister
				(inoAtHomePos:=GVL_iXlinker.Ec.EC.Ek.AB22.Channel_1.Input,
				inoAtWorkPos:=GVL_iXlinker.Ec.EC.Ek.AB22.Channel_2.Input,
				inoToHomePos:=tempBoolHome,
				inoToWorkPos:=tempBoolWork);
GVL_iXlinker.Ec.EC.Ek.PNEU.Modules.Outputs.digital_Data_O[2].1:=tempBoolHome;
GVL_iXlinker.Ec.EC.Ek.PNEU.Modules.Outputs.digital_Data_O[2].0:=tempBoolWork;

Components.PlsPaletizator.Components.P8_FixEntryBlisterSide
				(inoAtHomePos1:=GVL_iXlinker.Ec.EC.Ek.AB22.Channel_3.Input,
				inoAtWorkPos1:=GVL_iXlinker.Ec.EC.Ek.AB22.Channel_4.Input,
				inoAtHomePos2:=GVL_iXlinker.Ec.EC.Ek.AB22.Channel_5.Input,
				inoAtWorkPos2:=GVL_iXlinker.Ec.EC.Ek.AB22.Channel_6.Input,
				inoToHomePos:=tempBoolHome,
				inoToWorkPos:=tempBoolWork);
GVL_iXlinker.Ec.EC.Ek.PNEU.Modules.Outputs.digital_Data_O[2].3:=tempBoolHome;
GVL_iXlinker.Ec.EC.Ek.PNEU.Modules.Outputs.digital_Data_O[2].2:=tempBoolWork;

Components.PlsPaletizator(inSafeCondition:=GVL_iXlinker.Ec.EC.IA1.Channel_1.Input);
Components.PlsPaletizator.Service();
END_METHOD

(*~
	<docu>
		<summary>
			Controls `manual` mode of `CU00x`.
		</summary>
	</docu>
~*)
METHOD Manual : BOOL
VAR_INPUT
END_VAR
(*
	Enable condition to start `automatTask`.
	Modify according your needs.
	[! 
	THIS IS NOT SAFETY CONDITION. THE SAFETY OF PRESONNEL AND EQUIPMENT MUST BE ENSURED BY ADDITIONAL MEANS 
	TO COMPLY WITH REGULATIONS
	]
*)

	//_manualTask.Task.Enabled := THIS^.Technology.AllowManual();

	
(*
	or use default behavior from abstraction
*)
	SUPER^.Manual();
	

(*

	Executes sequence of manualTask.

*)
_manualTask();
END_METHOD

PROPERTY ManualTask : REFERENCE TO TcoTaskedService
GET
ManualTask REF= _manualTask;
END_GET
END_PROPERTY

PROPERTY ProductionPlanerTask : REFERENCE TO ProductionPlaner
GET
ProductionPlanerTask REF= _productionPlaner;
END_GET
END_PROPERTY

PROPERTY RecoverTask : REFERENCE TO CUBaseRecover
GET
RecoverTask REF= _recoverTask;
END_GET
END_PROPERTY

PROPERTY StatusInfo : REFERENCE TO CUBaseStatusInfo
GET
StatusInfo ref= _statusInfo;
END_GET
END_PROPERTY

PROPERTY SuspendTask : REFERENCE TO CUBaseSuspend
GET
SuspendTask REF= _suspendTask;
END_GET
END_PROPERTY

PROPERTY Technology : REFERENCE TO Technology
GET
VAR
    _technology : POINTER TO Technology;
END_VAR
IF __QUERYPOINTER(Parent, _technology) THEN // Check if _Parent is Station001
    Technology REF= _technology^;              // If the check is successful dereference a pointer. simlar to THIS^ or SUPER^
END_IF
END_GET
END_PROPERTY

END_FUNCTION_BLOCK

// ---- Technology/Technology.TcPOU
FUNCTION_BLOCK Technology EXTENDS TcoCore.TcoContext
VAR	
    _processSettings     : ProcessDataManager(THIS^);  			//a.k.a receipe
	_reworkSettings     : ProcessDataManager(THIS^);  			//a.k.a receipe for rework
    _technologySettings  : TechnologicalDataManager(THIS^);		//a.k.a machine settings
    _processTraceability : ProcessDataManager(THIS^);			//the same structure as process setting but filled with actual production data (measurements, inspection results, etc)
	
	
	fbGetCurTaskIndex            : GETCURTASKINDEX;
	_notificationPanel      : NotificationPanel(THIS^);				//provide technology state signals to side baner in visualisation
    {attribute addProperty Name "<#AUTOMAT ALL#>"}
    _automatAllTask : TcoCore.TcoTask(THIS^);					// Commmand-like taks to execute automation mode on whole technology. Handled in controlled units.
    {attribute addProperty Name "<#GROUND ALL#>"}
    _groundAllTask : TcoCore.TcoTask(THIS^);	

	{attribute addProperty Name "<#_cu00x#>"}					
    _cu00x         : CU00x(THIS^);
	
	{attribute addProperty Name "<#Technology Components#>"}	
	_components : TechnologyComponents:= (Parent := THIS^);

	{attribute addProperty Name "Device 1 (EtherCAT)"}
	Device_1 : TcoIo.TcoEthercatMasterDevice(THIS^);
	
	_setDummyConditionsSuffisient:BOOL;
	_dummyBlinker              : TcoUtilities.TcoBlinker(THIS^);
END_VAR

METHOD AllowAutomat : BOOL
VAR_INPUT
END_VAR
AllowAutomat := TRUE;
END_METHOD

METHOD AllowGround : BOOL
VAR_INPUT
END_VAR
AllowGround := TRUE;
END_METHOD

METHOD AllowManual :  BOOL
VAR_INPUT
END_VAR
AllowManual := TRUE;
END_METHOD

PROPERTY AutomatAllTask : REFERENCE TO TcoCore.TcoTask
GET
AutomatAllTask REF= _automatAllTask;
END_GET
END_PROPERTY

PROPERTY PUBLIC Cu00x : Reference to CU00x
GET
Cu00x REF=_cu00x;
END_GET
END_PROPERTY

METHOD ForceStepMode : BOOL
ForceStepMode := FALSE;
END_METHOD

PROPERTY GroundAllTask : REFERENCE TO TcoCore.TcoTask
GET
GroundAllTask REF= _groundAllTask;
END_GET
END_PROPERTY

METHOD InitializeComponents
VAR_INPUT
END_VAR

VAR
	controlVolage: BOOL;
	controlVoltageDoor: BOOL;
	estop: BOOL;
	presure: BOOL;
	locked: BOOL;
	lock: BOOL;
	opened: BOOL;
	closed: BOOL;
	
END_VAR
controlVolage:=FALSE;
controlVoltageDoor:=FALSE;
estop:=FALSE;
presure:=FALSE;

//_dummyBlinker(inOffTime := T#10000MS, inOnTime := T#10000MS);
(*
closed:=GVL_iXlinker.EC1.EK1200.IA1_EL1809.Channel_8.Input;
locked:=GVL_iXlinker.EC1.EK1200.IA1_EL1809.Channel_9.Input;

IF _setDummyConditionsSuffisient THEN
	controlVolage:=TRUE;
	controlVoltageDoor:=TRUE;
	estop:=FALSE;
	presure:=TRUE;


END_IF;

_components.ModeKey(inoKeyState1:=GVL_iXlinker.EC1.EK1200.IA1_EL1809.Channel_1.Input ,
					inoKeyState2:=GVL_iXlinker.EC1.EK1200.IA1_EL1809.Channel_2.Input);
					
_components.NormalServiceKey(inoSignal:=GVL_iXlinker.EC1.EK1200.IA1_EL1809.Channel_3.Input);
					
_components.ControlButtons(
	inoButtonRecover:=GVL_iXlinker.EC1.EK1200.IA1_EL1809.Channel_4.Input  , 
	inoButtonSuspend:=GVL_iXlinker.EC1.EK1200.IA1_EL1809.Channel_5.Input  , 
	inoButtonGround:=GVL_iXlinker.EC1.EK1200.IA1_EL1809.Channel_6.Input , 
	inoButtonAuto:=GVL_iXlinker.EC1.EK1200.IA1_EL1809.Channel_7.Input, 
	inoButtonRecoverLight:=GVL_iXlinker.EC1.EK1200.QA1_EL2809.Channel_1.Output  , 
	inoButtonSuspendLight:=GVL_iXlinker.EC1.EK1200.QA1_EL2809.Channel_2.Output  , 
	inoButtonGroundLight:=GVL_iXlinker.EC1.EK1200.QA1_EL2809.Channel_3.Output  , 
	inoButtonAutoLight:= GVL_iXlinker.EC1.EK1200.QA1_EL2809.Channel_4.Output );
	

					

_components.GlobalControlVoltage(inoSignal := controlVolage);

_components.LocalControlVoltage(inoSignal := controlVolage);
_components.LocalDoorVoltage(inoSignal := controlVoltageDoor);

_components.EmergencyStop(inoSignal := estop);
_components.AirPresureOk(inoSignal:= presure);


_components.StandardDoor(inoIsLocked := locked,
    inoIsOpen := opened,
    inoLock :=lock);
	
	
_components.BasicDoor(inoIsClosed := closed,
     inoLock := lock);


_components.DoorCicuit();

_components.Zone(inDoorCircuit:=_components.DoorCicuit,
				inEstopActive:=_components.EmergencyStop.Signal,
				inAirPressureOK:= _components.AirPresureOk.Signal);
		
				
_components.Zone.Service();
*)
END_METHOD

METHOD InitializeComponentsOnce
VAR_INPUT
END_VAR
_components.DoorCicuit.Restore();
_components.Zone.Restore();



_components.DoorCicuit.AddDoors(inDoor:=_components.StandardDoor);
_components.DoorCicuit.AddDoors(inDoor:=_components.BasicDoor);
_components.DoorCicuit.AddGlobalVoltage(inVoltage:=_components.GlobalControlVoltage);
_components.DoorCicuit.AddLocalVoltage(inVoltage:=_components.LocalControlVoltage);
_components.DoorCicuit.AddLocalDoorsVoltage(inVoltage:=_components.LocalDoorVoltage);


_components.Zone.AddControlledUnit(inControlledUnit:=_cu00x);
_components.Zone.AddControlButtons(inControlButtons:=_components.ControlButtons);
_components.Zone.AddKeyMode(inKeyMode:=_components.ModeKey);
_components.Zone.AddKeyNormalService(inKeyNormalService:=_components.NormalServiceKey);
END_METHOD

(*~
	<docu>
		<summary>
			Main method of the TcoContext. This is the entry point of any control logic that belongs to this context. 
			The call of this method is ensured by calling the <c>InstanceName.Run()</c> method, and it must not be called explicitly.
			This method is abstract, and it must be overridden in derived block.
		</summary>
	</docu>
~*)
METHOD PROTECTED Main
VAR
	_notificationSourceSignals: NotificationPanelInfo;
	safetyCircuitOk: BOOL;
	_eStopActive: BOOL;
	_keysAto: BOOL;
	_closed: BOOL;
	_locked: BOOL;
END_VAR
(*
	Context settings 
*)

// RTC Synchronisation
THIS^.RtcSynchronize(TRUE,  
					 '192.168.4.1.1.1',    // Provide AMS ID of the time source, leave blank if local. 
					 60);

// Messenger logger settings
_settings.Messaging.MessageDigestMethod := eMessageDigestMethod.CRC32;
_settings.Messaging.MessengerLoggingMethod := eMessengerLogMethod.OnEventRisen;


_components.DoorCicuit.Config.MaxDoors:=12;
_components.DoorCicuit.Config.MaxGlobalVoltage:=2;
_components.DoorCicuit.Config.MaxLocalVoltage:=2;
_components.DoorCicuit.Config.MaxLocalDoorsVoltage:=2;


_components.Zone.Config.MaxControlButtons:=2;
_components.Zone.Config.MaxControledUnits:=10;
_components.Zone.Config.MaxKeyMode:=2;
_components.Zone.Config.MaxKeyNormalService:=2;



THIS^.InitializeComponents();
fbGetCurTaskIndex();
IF _TaskInfo[fbGetCurTaskIndex.index].FirstCycle THEN
    // The code that you want to be executed at the first cycle of  PLC only 
	THIS^.InitializeComponentsOnce();
END_IF

//notification panel
 Context.Environment.Messaging.Suspend();
			
_closed:=TRUE;
//_closed   := 	Components.Safety.DoorCircuits.DoorCircuit_2.IsClosed 
//			AND Components.Safety.DoorCircuits.DoorCircuit_3.IsClosed  
//			AND Components.Safety.DoorCircuits.DoorCircuit_4.IsClosed  
//			AND Components.Safety.DoorCircuits.DoorCircuit_5.IsClosed  
//			AND Components.Safety.DoorCircuits.DoorCircuit_6.IsClosed;

 _locked:=TRUE;
//_locked   := 	Components.Safety.DoorCircuits.DoorCircuit_2.IsLocked 
//			AND Components.Safety.DoorCircuits.DoorCircuit_3.IsLocked  
//			AND Components.Safety.DoorCircuits.DoorCircuit_4.IsLocked  
//			AND Components.Safety.DoorCircuits.DoorCircuit_5.IsLocked  
//			AND Components.Safety.DoorCircuits.DoorCircuit_6.IsLocked;
			
_keysAto  := TRUE;
_eStopActive:=0;


_notificationSourceSignals.ControlVoltage   := TRUE;//Components.ControlVoltage.Signal.Signal 
_notificationSourceSignals.AirPressure      := TRUE;//Components.AirPressureOk.Signal.Signal, 
_notificationSourceSignals.AutomatAllowed   := _keysAto; 
_notificationSourceSignals.EmergencyStop    := _eStopActive > 0; 
_notificationSourceSignals.SafetyDoorOk     :=safetyCircuitOk;	
_notificationSourceSignals.LightCurtain     := TRUE; 	// not used
_notificationSourceSignals.DoorClosed       := _closed; 
_notificationSourceSignals.DoorLocked       := _locked; 
_notificationSourceSignals.ProcessDataOk    := _processSettings._data._EntityId <> '';
_notificationSourceSignals.TechnologyDataOk := _technologySettings._data._EntityId <> '';  
	
_notificationPanel(inBlinkPeriod:=T#500MS , inSignalSource:=_notificationSourceSignals );
			
 Context.Environment.Messaging.Resume();

(*
	
	Data managers

*)

_processSettings();
_reworkSettings();
_technologySettings();

(*

	Controlled units
	
*)

_cu00x();


_automatAllTask();
_groundAllTask();

//Device_1(	SyncUnits		:= ADR(		GVL_iXlinker.EC1.SyncUnits),
//			SyncUnitsSize	:= SIZEOF(	GVL_iXlinker.EC1.SyncUnits),
//			Inputs			:=			GVL_iXlinker.EC1.Inputs,
//			InfoData		:=			GVL_iXlinker.EC1.InfoData);
END_METHOD


(*~
	<docu>
		<summary>
			Called upon exit from the context. When overridden in derived class allows to execute an arbitrary logic after closing the context cycle.	
		</summary>			
	</docu>	
~*)METHOD PROTECTED OnExit
_automatAllTask.DoneWhen(TRUE);
_groundAllTask.DoneWhen(TRUE);
END_METHOD

PROPERTY ProcessSettings : REFERENCE TO ProcessDataManager
GET
ProcessSettings REF= _processSettings;
END_GET
END_PROPERTY

PROPERTY ReworkSettings : REFERENCE TO ProcessDataManager
GET
ReworkSettings REF= _reworkSettings;
END_GET
END_PROPERTY

PROPERTY TechnologicalSettings : REFERENCE TO TechnologicalDataManager
GET
TechnologicalSettings REF= _technologySettings;
END_GET
END_PROPERTY

END_FUNCTION_BLOCK
